LIN {X 0,Y 352.89,Z 1008.844,A -85,B 0,C 180,E1 14540.285,E2 14540.285} C_VEL
LIN {X 0,Y 348.435,Z 1029.036,A -85,B 0,C 180,E1 14538.872,E2 14538.872} C_VEL
LIN {X 0,Y 343.663,Z 1047.021,A -85,B 0,C 180,E1 14537.32,E2 14537.32} C_VEL
LIN {X 0,Y 338.159,Z 1064.954,A -85,B 0,C 180,E1 14535.444,E2 14535.444} C_VEL
LIN {X 0,Y 332.328,Z 1081.93,A -85,B 0,C 180,E1 14533.31,E2 14533.31} C_VEL
LIN {X 0,Y 326.202,Z 1097.954,A -85,B 0,C 180,E1 14530.873,E2 14530.873} C_VEL
LIN {X 0,Y 320.161,Z 1112.555,A -85,B 0,C 180,E1 14528.194,E2 14528.194} C_VEL
LIN {X 0,Y 314.194,Z 1126.284,A -85,B 0,C 180,E1 14525.168,E2 14525.168} C_VEL
LIN {X 0,Y 308.597,Z 1138.58,A -85,B 0,C 180,E1 14521.878,E2 14521.878} C_VEL
LIN {X 0,Y 303.562,Z 1149.432,A -85,B 0,C 180,E1 14518.313,E2 14518.313} C_VEL
LIN {X 0,Y 299.051,Z 1159.359,A -85,B 0,C 180,E1 14514.282,E2 14514.282} C_VEL
LIN {X 0,Y 295.723,Z 1167.059,A -85,B 0,C 180,E1 14510.38,E2 14510.38} C_VEL
LIN {X 0,Y 293.189,Z 1173.301,A -85,B 0,C 180,E1 14506.238,E2 14506.238} C_VEL
LIN {X 0,Y 291.464,Z 1178.188,A -85,B 0,C 180,E1 14501.878,E2 14501.878} C_VEL
LIN {X 0,Y 290.533,Z 1181.461,A -85,B 0,C 180,E1 14497.63,E2 14497.63} C_VEL
LIN {X 0,Y 290.087,Z 1183.156,A -85,B 0,C 180,E1 14493.557,E2 14493.557} C_VEL
LIN {X 0,Y 289.998,Z 1183.636,A -85,B 0,C 180,E1 14489.21,E2 14489.21} C_VEL
LIN {X 0,Y 290.174,Z 1182.841,A -85,B 0,C 180,E1 14485.257,E2 14485.257} C_VEL
LIN {X 0,Y 290.781,Z 1180.528,A -85,B 0,C 180,E1 14480.899,E2 14480.899} C_VEL
LIN {X 0,Y 291.906,Z 1176.965,A -85,B 0,C 180,E1 14476.733,E2 14476.733} C_VEL
LIN {X 0,Y 293.906,Z 1171.558,A -85,B 0,C 180,E1 14472.376,E2 14472.376} C_VEL
LIN {X 0,Y 296.703,Z 1164.7,A -85,B 0,C 180,E1 14468.243,E2 14468.243} C_VEL
LIN {X 0,Y 300.556,Z 1156.069,A -85,B 0,C 180,E1 14464.165,E2 14464.165} C_VEL
LIN {X 0,Y 305.239,Z 1146,A -85,B 0,C 180,E1 14460.356,E2 14460.356} C_VEL
LIN {X 0,Y 310.566,Z 1134.355,A -85,B 0,C 180,E1 14456.818,E2 14456.818} C_VEL
LIN {X 0,Y 316.433,Z 1121.267,A -85,B 0,C 180,E1 14453.557,E2 14453.557} C_VEL
LIN {X 0,Y 322.507,Z 1107.189,A -85,B 0,C 180,E1 14450.655,E2 14450.655} C_VEL
LIN {X 0,Y 328.545,Z 1092.152,A -85,B 0,C 180,E1 14448.089,E2 14448.089} C_VEL
LIN {X 0,Y 330.194,Z 1087.778,A -85,B 0,C 180,E1 14447.426,E2 14447.426} C_VEL
LIN {X 0,Y 331.529,Z 1082.425,A -85,B 0,C 180,E1 14446.505,E2 14446.505} C_VEL
LIN {X 0,Y 332.538,Z 1068.9,A -85,B 0,C 180,E1 14443.929,E2 14443.929} C_VEL
LIN {X 0,Y 333.902,Z 1062.973,A -85,B 0,C 180,E1 14443.095,E2 14443.095} C_VEL
LIN {X 0,Y 339.356,Z 1045.21,A -85,B 0,C 180,E1 14441.298,E2 14441.298} C_VEL
LIN {X 0,Y 344.539,Z 1025.743,A -85,B 0,C 180,E1 14439.676,E2 14439.676} C_VEL
LIN {X 0,Y 348.798,Z 1006.372,A -85,B 0,C 180,E1 14438.373,E2 14438.373} C_VEL
LIN {X 0,Y 352.358,Z 985.537,A -85,B 0,C 180,E1 14437.265,E2 14437.265} C_VEL
LIN {X 0,Y 355.126,Z 963.27,A -85,B 0,C 180,E1 14436.37,E2 14436.37} C_VEL
LIN {X 0,Y 356.788,Z 941.515,A -85,B 0,C 180,E1 14435.746,E2 14435.746} C_VEL
LIN {X 0,Y 365.568,Z 801.334,A -85,B 0,C 180,E1 14432.883,E2 14432.883} C_VEL
LIN {X 0,Y 356.931,Z 787.639,A -85,B 0,C 180,E1 14430.002,E2 14430.002} C_VEL
LIN {X 0,Y 349.574,Z 776.875,A -85,B 0,C 180,E1 14427.235,E2 14427.235} C_VEL
LIN {X 0,Y 343.426,Z 768.201,A -85,B 0,C 180,E1 14424.604,E2 14424.604} C_VEL
LIN {X 0,Y 339.11,Z 762.612,A -85,B 0,C 180,E1 14422.539,E2 14422.539} C_VEL
LIN {X 0,Y 335.486,Z 757.801,A -85,B 0,C 180,E1 14420.59,E2 14420.59} C_VEL
LIN {X 0,Y 331.948,Z 753.101,A -85,B 0,C 180,E1 14418.438,E2 14418.438} C_VEL
LIN {X 0,Y 328.093,Z 748.652,A -85,B 0,C 180,E1 14415.738,E2 14415.738} C_VEL
LIN {X 0,Y 327.083,Z 746.901,A -85,B 0,C 180,E1 14414.879,E2 14414.879} C_VEL
LIN {X 0,Y 323.777,Z 743.745,A -85,B 0,C 180,E1 14411.851,E2 14411.851} C_VEL
LIN {X 0,Y 322.352,Z 740.871,A -85,B 0,C 180,E1 14410.003,E2 14410.003} C_VEL
LIN {X 0,Y 318.916,Z 738.292,A -85,B 0,C 180,E1 14401.977,E2 14401.977} C_VEL
LIN {X 0,Y 319.479,Z 738.987,A -85,B 0,C 180,E1 14397.489,E2 14397.489} C_VEL
LIN {X 0,Y 322.551,Z 741.221,A -85,B 0,C 180,E1 14392.161,E2 14392.161} C_VEL
LIN {X 0,Y 324.789,Z 745.036,A -85,B 0,C 180,E1 14389.536,E2 14389.536} C_VEL
LIN {X 0,Y 325.775,Z 746.474,A -85,B 0,C 180,E1 14388.583,E2 14388.583} C_VEL
LIN {X 0,Y 329.072,Z 751.848,A -85,B 0,C 180,E1 14385.798,E2 14385.798} C_VEL
LIN {X 0,Y 332.186,Z 756.763,A -85,B 0,C 180,E1 14383.61,E2 14383.61} C_VEL
LIN {X 0,Y 337.821,Z 765.785,A -85,B 0,C 180,E1 14380.281,E2 14380.281} C_VEL
LIN {X 0,Y 345.029,Z 777.9,A -85,B 0,C 180,E1 14376.744,E2 14376.744} C_VEL
LIN {X 0,Y 351.975,Z 790.146,A -85,B 0,C 180,E1 14373.831,E2 14373.831} C_VEL
LIN {X 0,Y 359.361,Z 804.087,A -85,B 0,C 180,E1 14371.091,E2 14371.091} C_VEL
LIN {X 0,Y 365.817,Z 817.108,A -85,B 0,C 180,E1 14368.92,E2 14368.92} C_VEL
LIN {X 0,Y 356.497,Z 967.98,A -85,B 0,C 180,E1 14365.848,E2 14365.848} C_VEL
LIN {X 0,Y 352.635,Z 1028.021,A -85,B 0,C 180,E1 14364.593,E2 14364.593} C_VEL
LIN {X 0,Y 349.693,Z 1050.79,A -85,B 0,C 180,E1 14363.922,E2 14363.922} C_VEL
LIN {X 0,Y 345.509,Z 1072.869,A -85,B 0,C 180,E1 14363.073,E2 14363.073} C_VEL
LIN {X 0,Y 340.542,Z 1093.764,A -85,B 0,C 180,E1 14362.028,E2 14362.028} C_VEL
LIN {X 0,Y 334.973,Z 1113.773,A -85,B 0,C 180,E1 14360.721,E2 14360.721} C_VEL
LIN {X 0,Y 328.728,Z 1133.727,A -85,B 0,C 180,E1 14359.074,E2 14359.074} C_VEL
LIN {X 0,Y 322.404,Z 1152.314,A -85,B 0,C 180,E1 14357.187,E2 14357.187} C_VEL
LIN {X 0,Y 315.474,Z 1171.079,A -85,B 0,C 180,E1 14354.843,E2 14354.843} C_VEL
LIN {X 0,Y 308.833,Z 1188.354,A -85,B 0,C 180,E1 14352.204,E2 14352.204} C_VEL
LIN {X 0,Y 302.39,Z 1204.876,A -85,B 0,C 180,E1 14349.163,E2 14349.163} C_VEL
LIN {X 0,Y 296.695,Z 1219.605,A -85,B 0,C 180,E1 14345.899,E2 14345.899} C_VEL
LIN {X 0,Y 291.735,Z 1233.031,A -85,B 0,C 180,E1 14342.319,E2 14342.319} C_VEL
LIN {X 0,Y 287.46,Z 1245.829,A -85,B 0,C 180,E1 14338.231,E2 14338.231} C_VEL
LIN {X 0,Y 284.419,Z 1256.619,A -85,B 0,C 180,E1 14334.065,E2 14334.065} C_VEL
LIN {X 0,Y 282.517,Z 1265.437,A -85,B 0,C 180,E1 14329.861,E2 14329.861} C_VEL
LIN {X 0,Y 281.556,Z 1272.909,A -85,B 0,C 180,E1 14325.446,E2 14325.446} C_VEL
LIN {X 0,Y 281.384,Z 1278.064,A -85,B 0,C 180,E1 14321.477,E2 14321.477} C_VEL
LIN {X 0,Y 281.608,Z 1281.89,A -85,B 0,C 180,E1 14317.343,E2 14317.343} C_VEL
LIN {X 0,Y 281.909,Z 1283.834,A -85,B 0,C 180,E1 14313.864,E2 14313.864} C_VEL
LIN {X 0,Y 282.055,Z 1284.645,A -85,B 0,C 180,E1 14310.203,E2 14310.203} C_VEL
LIN {X 0,Y 281.933,Z 1283.994,A -85,B 0,C 180,E1 14306.544,E2 14306.544} C_VEL
LIN {X 0,Y 281.649,Z 1282.161,A -85,B 0,C 180,E1 14303.068,E2 14303.068} C_VEL
LIN {X 0,Y 281.387,Z 1278.535,A -85,B 0,C 180,E1 14298.938,E2 14298.938} C_VEL
LIN {X 0,Y 281.512,Z 1273.495,A -85,B 0,C 180,E1 14294.973,E2 14294.973} C_VEL
LIN {X 0,Y 282.383,Z 1266.228,A -85,B 0,C 180,E1 14290.56,E2 14290.56} C_VEL
LIN {X 0,Y 284.184,Z 1257.547,A -85,B 0,C 180,E1 14286.354,E2 14286.354} C_VEL
LIN {X 0,Y 287.105,Z 1246.946,A -85,B 0,C 180,E1 14282.183,E2 14282.183} C_VEL
LIN {X 0,Y 291.426,Z 1233.864,A -85,B 0,C 180,E1 14277.933,E2 14277.933} C_VEL
LIN {X 0,Y 296.389,Z 1220.386,A -85,B 0,C 180,E1 14274.296,E2 14274.296} C_VEL
LIN {X 0,Y 302.022,Z 1205.722,A -85,B 0,C 180,E1 14271.025,E2 14271.025} C_VEL
LIN {X 0,Y 308.619,Z 1188.814,A -85,B 0,C 180,E1 14267.885,E2 14267.885} C_VEL
LIN {X 0,Y 315.232,Z 1171.616,A -85,B 0,C 180,E1 14265.241,E2 14265.241} C_VEL
LIN {X 0,Y 321.854,Z 1153.662,A -85,B 0,C 180,E1 14262.982,E2 14262.982} C_VEL
LIN {X 0,Y 328.49,Z 1134.282,A -85,B 0,C 180,E1 14260.989,E2 14260.989} C_VEL
LIN {X 0,Y 334.765,Z 1114.287,A -85,B 0,C 180,E1 14259.327,E2 14259.327} C_VEL
LIN {X 0,Y 340.532,Z 1093.545,A -85,B 0,C 180,E1 14257.97,E2 14257.97} C_VEL
LIN {X 0,Y 345.5,Z 1072.584,A -85,B 0,C 180,E1 14256.924,E2 14256.924} C_VEL
LIN {X 0,Y 349.774,Z 1049.728,A -85,B 0,C 180,E1 14256.053,E2 14256.053} C_VEL
LIN {X 0,Y 352.628,Z 1027.173,A -85,B 0,C 180,E1 14255.396,E2 14255.396} C_VEL
LIN {X 0,Y 359.75,Z 913.323,A -85,B 0,C 180,E1 14253.052,E2 14253.052} C_VEL
LIN {X 0,Y 365.721,Z 817.058,A -85,B 0,C 180,E1 14251.089,E2 14251.089} C_VEL
LIN {X 0,Y 357.817,Z 801.163,A -85,B 0,C 180,E1 14248.407,E2 14248.407} C_VEL
LIN {X 0,Y 350.738,Z 788.072,A -85,B 0,C 180,E1 14245.736,E2 14245.736} C_VEL
LIN {X 0,Y 343.692,Z 775.733,A -85,B 0,C 180,E1 14242.717,E2 14242.717} C_VEL
LIN {X 0,Y 337.149,Z 764.789,A -85,B 0,C 180,E1 14239.444,E2 14239.444} C_VEL
LIN {X 0,Y 331.093,Z 755.02,A -85,B 0,C 180,E1 14235.77,E2 14235.77} C_VEL
LIN {X 0,Y 327.647,Z 749.717,A -85,B 0,C 180,E1 14233.23,E2 14233.23} C_VEL
LIN {X 0,Y 324.965,Z 745.249,A -85,B 0,C 180,E1 14230.817,E2 14230.817} C_VEL
LIN {X 0,Y 322.548,Z 741.379,A -85,B 0,C 180,E1 14228.108,E2 14228.108} C_VEL
LIN {X 0,Y 322.074,Z 740.745,A -85,B 0,C 180,E1 14227.492,E2 14227.492} C_VEL
LIN {X 0,Y 318.696,Z 738.017,A -85,B 0,C 180,E1 14219.64,E2 14219.64} C_VEL
LIN {X 0,Y 319.045,Z 738.532,A -85,B 0,C 180,E1 14215.686,E2 14215.686} C_VEL
LIN {X 0,Y 322.489,Z 741.155,A -85,B 0,C 180,E1 14209.459,E2 14209.459} C_VEL
LIN {X 0,Y 324.685,Z 744.973,A -85,B 0,C 180,E1 14206.918,E2 14206.918} C_VEL
LIN {X 0,Y 327.369,Z 747.393,A -85,B 0,C 180,E1 14204.635,E2 14204.635} C_VEL
LIN {X 0,Y 330.353,Z 751.615,A -85,B 0,C 180,E1 14202.382,E2 14202.382} C_VEL
LIN {X 0,Y 332.04,Z 753.353,A -85,B 0,C 180,E1 14201.294,E2 14201.294} C_VEL
LIN {X 0,Y 335.636,Z 757.967,A -85,B 0,C 180,E1 14199.146,E2 14199.146} C_VEL
LIN {X 0,Y 341,Z 765.139,A -85,B 0,C 180,E1 14196.361,E2 14196.361} C_VEL
LIN {X 0,Y 345.217,Z 770.847,A -85,B 0,C 180,E1 14194.434,E2 14194.434} C_VEL
LIN {X 0,Y 350.999,Z 778.969,A -85,B 0,C 180,E1 14192.057,E2 14192.057} C_VEL
LIN {X 0,Y 359.038,Z 790.932,A -85,B 0,C 180,E1 14189.129,E2 14189.129} C_VEL
LIN {X 0,Y 365.542,Z 801.506,A -85,B 0,C 180,E1 14186.993,E2 14186.993} C_VEL
LIN {X 0,Y 356.293,Z 947.507,A -85,B 0,C 180,E1 14184.004,E2 14184.004} C_VEL
LIN {X 0,Y 354.431,Z 969.192,A -85,B 0,C 180,E1 14183.324,E2 14183.324} C_VEL
LIN {X 0,Y 351.586,Z 990.18,A -85,B 0,C 180,E1 14182.413,E2 14182.413} C_VEL
LIN {X 0,Y 347.909,Z 1010.243,A -85,B 0,C 180,E1 14181.283,E2 14181.283} C_VEL
LIN {X 0,Y 343.562,Z 1029.462,A -85,B 0,C 180,E1 14179.941,E2 14179.941} C_VEL
LIN {X 0,Y 338.513,Z 1047.906,A -85,B 0,C 180,E1 14178.35,E2 14178.35} C_VEL
LIN {X 0,Y 332.67,Z 1066.352,A -85,B 0,C 180,E1 14176.412,E2 14176.412} C_VEL
LIN {X 0,Y 326.549,Z 1083.514,A -85,B 0,C 180,E1 14174.235,E2 14174.235} C_VEL
LIN {X 0,Y 320.261,Z 1099.348,A -85,B 0,C 180,E1 14171.801,E2 14171.801} C_VEL
LIN {X 0,Y 313.967,Z 1113.957,A -85,B 0,C 180,E1 14169.089,E2 14169.089} C_VEL
LIN {X 0,Y 307.655,Z 1127.852,A -85,B 0,C 180,E1 14165.978,E2 14165.978} C_VEL
LIN {X 0,Y 301.87,Z 1139.986,A -85,B 0,C 180,E1 14162.675,E2 14162.675} C_VEL
LIN {X 0,Y 296.579,Z 1150.838,A -85,B 0,C 180,E1 14159.042,E2 14159.042} C_VEL
LIN {X 0,Y 291.81,Z 1160.765,A -85,B 0,C 180,E1 14154.925,E2 14154.925} C_VEL
LIN {X 0,Y 288.272,Z 1168.465,A -85,B 0,C 180,E1 14150.931,E2 14150.931} C_VEL
LIN {X 0,Y 285.565,Z 1174.705,A -85,B 0,C 180,E1 14146.684,E2 14146.684} C_VEL
LIN {X 0,Y 283.709,Z 1179.588,A -85,B 0,C 180,E1 14142.207,E2 14142.207} C_VEL
LIN {X 0,Y 282.715,Z 1182.813,A -85,B 0,C 180,E1 14137.928,E2 14137.928} C_VEL
LIN {X 0,Y 282.217,Z 1184.547,A -85,B 0,C 180,E1 14133.656,E2 14133.656} C_VEL
LIN {X 0,Y 282.12,Z 1185.026,A -85,B 0,C 180,E1 14129.188,E2 14129.188} C_VEL
LIN {X 0,Y 282.313,Z 1184.233,A -85,B 0,C 180,E1 14125.124,E2 14125.124} C_VEL
LIN {X 0,Y 282.972,Z 1181.924,A -85,B 0,C 180,E1 14120.646,E2 14120.646} C_VEL
LIN {X 0,Y 284.187,Z 1178.365,A -85,B 0,C 180,E1 14116.366,E2 14116.366} C_VEL
LIN {X 0,Y 286.33,Z 1172.962,A -85,B 0,C 180,E1 14111.894,E2 14111.894} C_VEL
LIN {X 0,Y 289.32,Z 1166.104,A -85,B 0,C 180,E1 14107.658,E2 14107.658} C_VEL
LIN {X 0,Y 293.405,Z 1157.474,A -85,B 0,C 180,E1 14103.487,E2 14103.487} C_VEL
LIN {X 0,Y 298.34,Z 1147.404,A -85,B 0,C 180,E1 14099.599,E2 14099.599} C_VEL
LIN {X 0,Y 303.948,Z 1135.742,A -85,B 0,C 180,E1 14095.994,E2 14095.994} C_VEL
LIN {X 0,Y 310.08,Z 1122.666,A -85,B 0,C 180,E1 14092.686,E2 14092.686} C_VEL
LIN {X 0,Y 316.419,Z 1108.584,A -85,B 0,C 180,E1 14089.746,E2 14089.746} C_VEL
LIN {X 0,Y 322.699,Z 1093.545,A -85,B 0,C 180,E1 14087.15,E2 14087.15} C_VEL
LIN {X 0,Y 328.977,Z 1077.07,A -85,B 0,C 180,E1 14084.799,E2 14084.799} C_VEL
LIN {X 0,Y 333.902,Z 1062.973,A -85,B 0,C 180,E1 14083.095,E2 14083.095} C_VEL
LIN {X 0,Y 335.311,Z 1056.946,A -85,B 0,C 180,E1 14082.291,E2 14082.291} C_VEL
LIN {X 0,Y 336.215,Z 1041.964,A -85,B 0,C 180,E1 14080.007,E2 14080.007} C_VEL
LIN {X 0,Y 337.38,Z 1035.478,A -85,B 0,C 180,E1 14079.315,E2 14079.315} C_VEL
LIN {X 0,Y 342.109,Z 1016.487,A -85,B 0,C 180,E1 14077.9,E2 14077.9} C_VEL
LIN {X 0,Y 345.996,Z 997.035,A -85,B 0,C 180,E1 14076.741,E2 14076.741} C_VEL
LIN {X 0,Y 349.241,Z 975.642,A -85,B 0,C 180,E1 14075.743,E2 14075.743} C_VEL
LIN {X 0,Y 351.436,Z 954.76,A -85,B 0,C 180,E1 14075.015,E2 14075.015} C_VEL
LIN {X 0,Y 353.764,Z 917.385,A -85,B 0,C 180,E1 14074.155,E2 14074.155} C_VEL
LIN {X 0,Y 361.124,Z 805.509,A -85,B 0,C 180,E1 14071.88,E2 14071.88} C_VEL
LIN {X 0,Y 352.872,Z 792.375,A -85,B 0,C 180,E1 14068.982,E2 14068.982} C_VEL
LIN {X 0,Y 344.727,Z 780.224,A -85,B 0,C 180,E1 14065.698,E2 14065.698} C_VEL
LIN {X 0,Y 337.992,Z 770.862,A -85,B 0,C 180,E1 14062.526,E2 14062.526} C_VEL
LIN {X 0,Y 333.504,Z 765.063,A -85,B 0,C 180,E1 14060.077,E2 14060.077} C_VEL
LIN {X 0,Y 329.693,Z 760.015,A -85,B 0,C 180,E1 14057.654,E2 14057.654} C_VEL
LIN {X 0,Y 326.481,Z 756.026,A -85,B 0,C 180,E1 14055.271,E2 14055.271} C_VEL
LIN {X 0,Y 325.482,Z 754.519,A -85,B 0,C 180,E1 14054.408,E2 14054.408} C_VEL
LIN {X 0,Y 322.268,Z 751.064,A -85,B 0,C 180,E1 14051.272,E2 14051.272} C_VEL
LIN {X 0,Y 321.105,Z 748.705,A -85,B 0,C 180,E1 14049.68,E2 14049.68} C_VEL
LIN {X 0,Y 317.941,Z 746.234,A -85,B 0,C 180,E1 14041.983,E2 14041.983} C_VEL
LIN {X 0,Y 318.504,Z 746.942,A -85,B 0,C 180,E1 14037.481,E2 14037.481} C_VEL
LIN {X 0,Y 321.362,Z 749.076,A -85,B 0,C 180,E1 14032.402,E2 14032.402} C_VEL
LIN {X 0,Y 323.635,Z 752.927,A -85,B 0,C 180,E1 14029.678,E2 14029.678} C_VEL
LIN {X 0,Y 325.216,Z 755.754,A -85,B 0,C 180,E1 14028.113,E2 14028.113} C_VEL
LIN {X 0,Y 327.462,Z 759.302,A -85,B 0,C 180,E1 14026.222,E2 14026.222} C_VEL
LIN {X 0,Y 330.543,Z 764.349,A -85,B 0,C 180,E1 14023.977,E2 14023.977} C_VEL
LIN {X 0,Y 335.976,Z 773.309,A -85,B 0,C 180,E1 14020.666,E2 14020.666} C_VEL
LIN {X 0,Y 342.612,Z 784.779,A -85,B 0,C 180,E1 14017.298,E2 14017.298} C_VEL
LIN {X 0,Y 349.295,Z 796.876,A -85,B 0,C 180,E1 14014.391,E2 14014.391} C_VEL
LIN {X 0,Y 356.412,Z 810.672,A -85,B 0,C 180,E1 14011.654,E2 14011.654} C_VEL
LIN {X 0,Y 361.421,Z 821.196,A -85,B 0,C 180,E1 14009.887,E2 14009.887} C_VEL
LIN {X 0,Y 348.204,Z 1024.194,A -85,B 0,C 180,E1 14005.738,E2 14005.738} C_VEL
LIN {X 0,Y 345.397,Z 1046.631,A -85,B 0,C 180,E1 14005.1,E2 14005.1} C_VEL
LIN {X 0,Y 341.208,Z 1069.196,A -85,B 0,C 180,E1 14004.26,E2 14004.26} C_VEL
LIN {X 0,Y 336.237,Z 1089.948,A -85,B 0,C 180,E1 14003.262,E2 14003.262} C_VEL
LIN {X 0,Y 330.546,Z 1109.941,A -85,B 0,C 180,E1 14001.995,E2 14001.995} C_VEL
LIN {X 0,Y 323.709,Z 1131.293,A -85,B 0,C 180,E1 14000.271,E2 14000.271} C_VEL
LIN {X 0,Y 317.051,Z 1150.222,A -85,B 0,C 180,E1 13998.364,E2 13998.364} C_VEL
LIN {X 0,Y 309.857,Z 1168.972,A -85,B 0,C 180,E1 13996.018,E2 13996.018} C_VEL
LIN {X 0,Y 302.883,Z 1186.338,A -85,B 0,C 180,E1 13993.363,E2 13993.363} C_VEL
LIN {X 0,Y 296.281,Z 1202.484,A -85,B 0,C 180,E1 13990.385,E2 13990.385} C_VEL
LIN {X 0,Y 290.223,Z 1217.286,A -85,B 0,C 180,E1 13987.076,E2 13987.076} C_VEL
LIN {X 0,Y 284.73,Z 1231.282,A -85,B 0,C 180,E1 13983.306,E2 13983.306} C_VEL
LIN {X 0,Y 280.255,Z 1243.769,A -85,B 0,C 180,E1 13979.259,E2 13979.259} C_VEL
LIN {X 0,Y 276.924,Z 1254.627,A -85,B 0,C 180,E1 13974.988,E2 13974.988} C_VEL
LIN {X 0,Y 274.799,Z 1263.568,A -85,B 0,C 180,E1 13970.666,E2 13970.666} C_VEL
LIN {X 0,Y 273.67,Z 1271.159,A -85,B 0,C 180,E1 13966.12,E2 13966.12} C_VEL
LIN {X 0,Y 273.441,Z 1276.389,A -85,B 0,C 180,E1 13962.03,E2 13962.03} C_VEL
LIN {X 0,Y 273.659,Z 1280.338,A -85,B 0,C 180,E1 13957.769,E2 13957.769} C_VEL
LIN {X 0,Y 273.999,Z 1282.355,A -85,B 0,C 180,E1 13954.185,E2 13954.185} C_VEL
LIN {X 0,Y 274.169,Z 1283.18,A -85,B 0,C 180,E1 13950.836,E2 13950.836} C_VEL
LIN {X 0,Y 274.077,Z 1282.839,A -85,B 0,C 180,E1 13947.073,E2 13947.073} C_VEL
LIN {X 0,Y 273.767,Z 1281.029,A -85,B 0,C 180,E1 13943.289,E2 13943.289} C_VEL
LIN {X 0,Y 273.465,Z 1277.766,A -85,B 0,C 180,E1 13939.254,E2 13939.254} C_VEL
LIN {X 0,Y 273.557,Z 1272.643,A -85,B 0,C 180,E1 13934.96,E2 13934.96} C_VEL
LIN {X 0,Y 274.364,Z 1265.972,A -85,B 0,C 180,E1 13930.633,E2 13930.633} C_VEL
LIN {X 0,Y 276.17,Z 1257.449,A -85,B 0,C 180,E1 13926.306,E2 13926.306} C_VEL
LIN {X 0,Y 279.311,Z 1246.603,A -85,B 0,C 180,E1 13921.803,E2 13921.803} C_VEL
LIN {X 0,Y 283.361,Z 1234.976,A -85,B 0,C 180,E1 13917.805,E2 13917.805} C_VEL
LIN {X 0,Y 288.625,Z 1221.215,A -85,B 0,C 180,E1 13913.921,E2 13913.921} C_VEL
LIN {X 0,Y 294.763,Z 1206.044,A -85,B 0,C 180,E1 13910.38,E2 13910.38} C_VEL
LIN {X 0,Y 301.363,Z 1190.014,A -85,B 0,C 180,E1 13907.276,E2 13907.276} C_VEL
LIN {X 0,Y 308.16,Z 1173.152,A -85,B 0,C 180,E1 13904.58,E2 13904.58} C_VEL
LIN {X 0,Y 315.186,Z 1154.974,A -85,B 0,C 180,E1 13902.209,E2 13902.209} C_VEL
LIN {X 0,Y 322.281,Z 1135.335,A -85,B 0,C 180,E1 13900.117,E2 13900.117} C_VEL
LIN {X 0,Y 328.766,Z 1115.703,A -85,B 0,C 180,E1 13898.434,E2 13898.434} C_VEL
LIN {X 0,Y 334.613,Z 1095.56,A -85,B 0,C 180,E1 13897.08,E2 13897.08} C_VEL
LIN {X 0,Y 340.185,Z 1073.394,A -85,B 0,C 180,E1 13895.932,E2 13895.932} C_VEL
LIN {X 0,Y 344.585,Z 1051.413,A -85,B 0,C 180,E1 13895.066,E2 13895.066} C_VEL
LIN {X 0,Y 347.631,Z 1028.996,A -85,B 0,C 180,E1 13894.394,E2 13894.394} C_VEL
LIN {X 0,Y 350.084,Z 995.699,A -85,B 0,C 180,E1 13893.665,E2 13893.665} C_VEL
LIN {X 0,Y 361.293,Z 820.87,A -85,B 0,C 180,E1 13890.106,E2 13890.106} C_VEL
LIN {X 0,Y 353.804,Z 805.57,A -85,B 0,C 180,E1 13887.428,E2 13887.428} C_VEL
LIN {X 0,Y 346.866,Z 792.534,A -85,B 0,C 180,E1 13884.661,E2 13884.661} C_VEL
LIN {X 0,Y 340.077,Z 780.45,A -85,B 0,C 180,E1 13881.562,E2 13881.562} C_VEL
LIN {X 0,Y 334.728,Z 771.416,A -85,B 0,C 180,E1 13878.73,E2 13878.73} C_VEL
LIN {X 0,Y 329.477,Z 762.556,A -85,B 0,C 180,E1 13875.398,E2 13875.398} C_VEL
LIN {X 0,Y 326.023,Z 757.116,A -85,B 0,C 180,E1 13872.756,E2 13872.756} C_VEL
LIN {X 0,Y 323.623,Z 752.949,A -85,B 0,C 180,E1 13870.503,E2 13870.503} C_VEL
LIN {X 0,Y 321.233,Z 748.915,A -85,B 0,C 180,E1 13867.691,E2 13867.691} C_VEL
LIN {X 0,Y 317.751,Z 746.016,A -85,B 0,C 180,E1 13860,E2 13860} C_VEL
LIN {X 0,Y 317.91,Z 746.263,A -85,B 0,C 180,E1 13856.393,E2 13856.393} C_VEL
LIN {X 0,Y 321.298,Z 749.039,A -85,B 0,C 180,E1 13849.692,E2 13849.692} C_VEL
LIN {X 0,Y 323.447,Z 752.777,A -85,B 0,C 180,E1 13847.14,E2 13847.14} C_VEL
LIN {X 0,Y 325.919,Z 755.057,A -85,B 0,C 180,E1 13844.975,E2 13844.975} C_VEL
LIN {X 0,Y 328.951,Z 759.365,A -85,B 0,C 180,E1 13842.628,E2 13842.628} C_VEL
LIN {X 0,Y 330.476,Z 761.049,A -85,B 0,C 180,E1 13841.614,E2 13841.614} C_VEL
LIN {X 0,Y 334.864,Z 766.905,A -85,B 0,C 180,E1 13838.958,E2 13838.958} C_VEL
LIN {X 0,Y 339.197,Z 772.762,A -85,B 0,C 180,E1 13836.688,E2 13836.688} C_VEL
LIN {X 0,Y 344.785,Z 780.37,A -85,B 0,C 180,E1 13834.123,E2 13834.123} C_VEL
LIN {X 0,Y 353.678,Z 793.642,A -85,B 0,C 180,E1 13830.58,E2 13830.58} C_VEL
LIN {X 0,Y 361.1,Z 805.724,A -85,B 0,C 180,E1 13827.99,E2 13827.99} C_VEL
LIN {X 0,Y 351.736,Z 948.502,A -85,B 0,C 180,E1 13825.057,E2 13825.057} C_VEL
LIN {X 0,Y 349.827,Z 970.215,A -85,B 0,C 180,E1 13824.375,E2 13824.375} C_VEL
LIN {X 0,Y 346.884,Z 991.265,A -85,B 0,C 180,E1 13823.46,E2 13823.46} C_VEL
LIN {X 0,Y 343.038,Z 1011.641,A -85,B 0,C 180,E1 13822.309,E2 13822.309} C_VEL
LIN {X 0,Y 338.545,Z 1030.859,A -85,B 0,C 180,E1 13820.961,E2 13820.961} C_VEL
LIN {X 0,Y 333.333,Z 1049.278,A -85,B 0,C 180,E1 13819.365,E2 13819.365} C_VEL
LIN {X 0,Y 327.279,Z 1067.749,A -85,B 0,C 180,E1 13817.413,E2 13817.413} C_VEL
LIN {X 0,Y 321.012,Z 1084.726,A -85,B 0,C 180,E1 13815.246,E2 13815.246} C_VEL
LIN {X 0,Y 314.622,Z 1100.229,A -85,B 0,C 180,E1 13812.849,E2 13812.849} C_VEL
LIN {X 0,Y 307.854,Z 1115.359,A -85,B 0,C 180,E1 13810.02,E2 13810.02} C_VEL
LIN {X 0,Y 301.332,Z 1129.121,A -85,B 0,C 180,E1 13806.901,E2 13806.901} C_VEL
LIN {X 0,Y 295.206,Z 1141.392,A -85,B 0,C 180,E1 13803.509,E2 13803.509} C_VEL
LIN {X 0,Y 289.644,Z 1152.245,A -85,B 0,C 180,E1 13799.807,E2 13799.807} C_VEL
LIN {X 0,Y 284.605,Z 1162.173,A -85,B 0,C 180,E1 13795.601,E2 13795.601} C_VEL
LIN {X 0,Y 280.852,Z 1169.871,A -85,B 0,C 180,E1 13791.511,E2 13791.511} C_VEL
LIN {X 0,Y 277.957,Z 1176.109,A -85,B 0,C 180,E1 13787.155,E2 13787.155} C_VEL
LIN {X 0,Y 275.964,Z 1180.988,A -85,B 0,C 180,E1 13782.555,E2 13782.555} C_VEL
LIN {X 0,Y 274.887,Z 1184.209,A -85,B 0,C 180,E1 13778.155,E2 13778.155} C_VEL
LIN {X 0,Y 274.348,Z 1185.939,A -85,B 0,C 180,E1 13773.761,E2 13773.761} C_VEL
LIN {X 0,Y 274.242,Z 1186.417,A -85,B 0,C 180,E1 13769.164,E2 13769.164} C_VEL
LIN {X 0,Y 274.452,Z 1185.625,A -85,B 0,C 180,E1 13764.984,E2 13764.984} C_VEL
LIN {X 0,Y 275.167,Z 1183.32,A -85,B 0,C 180,E1 13760.378,E2 13760.378} C_VEL
LIN {X 0,Y 276.476,Z 1179.766,A -85,B 0,C 180,E1 13755.978,E2 13755.978} C_VEL
LIN {X 0,Y 278.647,Z 1174.633,A -85,B 0,C 180,E1 13751.593,E2 13751.593} C_VEL
LIN {X 0,Y 281.79,Z 1167.874,A -85,B 0,C 180,E1 13747.248,E2 13747.248} C_VEL
LIN {X 0,Y 285.952,Z 1159.588,A -85,B 0,C 180,E1 13743.08,E2 13743.08} C_VEL
LIN {X 0,Y 290.93,Z 1149.874,A -85,B 0,C 180,E1 13739.199,E2 13739.199} C_VEL
LIN {X 0,Y 296.711,Z 1138.458,A -85,B 0,C 180,E1 13735.521,E2 13735.521} C_VEL
LIN {X 0,Y 303.053,Z 1125.647,A -85,B 0,C 180,E1 13732.146,E2 13732.146} C_VEL
LIN {X 0,Y 309.793,Z 1111.407,A -85,B 0,C 180,E1 13729.068,E2 13729.068} C_VEL
LIN {X 0,Y 316.525,Z 1095.904,A -85,B 0,C 180,E1 13726.335,E2 13726.335} C_VEL
LIN {X 0,Y 323.231,Z 1079.068,A -85,B 0,C 180,E1 13723.886,E2 13723.886} C_VEL
LIN {X 0,Y 329.376,Z 1061.96,A -85,B 0,C 180,E1 13721.822,E2 13721.822} C_VEL
LIN {X 0,Y 334.988,Z 1043.996,A -85,B 0,C 180,E1 13720.043,E2 13720.043} C_VEL
LIN {X 0,Y 337.38,Z 1035.478,A -85,B 0,C 180,E1 13719.315,E2 13719.315} C_VEL
LIN {X 0,Y 338.592,Z 1028.887,A -85,B 0,C 180,E1 13718.645,E2 13718.645} C_VEL
LIN {X 0,Y 339.096,Z 1012.653,A -85,B 0,C 180,E1 13716.637,E2 13716.637} C_VEL
LIN {X 0,Y 339.952,Z 1005.7,A -85,B 0,C 180,E1 13716.083,E2 13716.083} C_VEL
LIN {X 0,Y 343.561,Z 985.118,A -85,B 0,C 180,E1 13715.02,E2 13715.02} C_VEL
LIN {X 0,Y 346.205,Z 963.954,A -85,B 0,C 180,E1 13714.195,E2 13714.195} C_VEL
LIN {X 0,Y 347.99,Z 940.649,A -85,B 0,C 180,E1 13713.548,E2 13713.548} C_VEL
LIN {X 0,Y 356.777,Z 809.833,A -85,B 0,C 180,E1 13710.854,E2 13710.854} C_VEL
LIN {X 0,Y 349.5,Z 798.065,A -85,B 0,C 180,E1 13708.167,E2 13708.167} C_VEL
LIN {X 0,Y 342.23,Z 787.038,A -85,B 0,C 180,E1 13705.111,E2 13705.111} C_VEL
LIN {X 0,Y 335.916,Z 778.069,A -85,B 0,C 180,E1 13702.027,E2 13702.027} C_VEL
LIN {X 0,Y 331.69,Z 772.464,A -85,B 0,C 180,E1 13699.64,E2 13699.64} C_VEL
LIN {X 0,Y 328.105,Z 767.601,A -85,B 0,C 180,E1 13697.285,E2 13697.285} C_VEL
LIN {X 0,Y 324.89,Z 763.4,A -85,B 0,C 180,E1 13694.8,E2 13694.8} C_VEL
LIN {X 0,Y 324.109,Z 762.262,A -85,B 0,C 180,E1 13694.106,E2 13694.106} C_VEL
LIN {X 0,Y 320.997,Z 758.758,A -85,B 0,C 180,E1 13690.953,E2 13690.953} C_VEL
LIN {X 0,Y 320.003,Z 756.6,A -85,B 0,C 180,E1 13689.532,E2 13689.532} C_VEL
LIN {X 0,Y 316.967,Z 754.176,A -85,B 0,C 180,E1 13681.989,E2 13681.989} C_VEL
LIN {X 0,Y 317.472,Z 754.834,A -85,B 0,C 180,E1 13677.654,E2 13677.654} C_VEL
LIN {X 0,Y 320.18,Z 756.923,A -85,B 0,C 180,E1 13672.644,E2 13672.644} C_VEL
LIN {X 0,Y 322.483,Z 760.818,A -85,B 0,C 180,E1 13669.821,E2 13669.821} C_VEL
LIN {X 0,Y 326.025,Z 767.05,A -85,B 0,C 180,E1 13666.522,E2 13666.522} C_VEL
LIN {X 0,Y 328.855,Z 771.819,A -85,B 0,C 180,E1 13664.391,E2 13664.391} C_VEL
LIN {X 0,Y 334.146,Z 780.832,A -85,B 0,C 180,E1 13661.055,E2 13661.055} C_VEL
LIN {X 0,Y 340.389,Z 791.976,A -85,B 0,C 180,E1 13657.779,E2 13657.779} C_VEL
LIN {X 0,Y 346.649,Z 803.604,A -85,B 0,C 180,E1 13654.959,E2 13654.959} C_VEL
LIN {X 0,Y 353.597,Z 817.449,A -85,B 0,C 180,E1 13652.189,E2 13652.189} C_VEL
LIN {X 0,Y 357.053,Z 825.011,A -85,B 0,C 180,E1 13650.908,E2 13650.908} C_VEL
LIN {X 0,Y 343.648,Z 1023.437,A -85,B 0,C 180,E1 13646.841,E2 13646.841} C_VEL
LIN {X 0,Y 340.733,Z 1045.78,A -85,B 0,C 180,E1 13646.2,E2 13646.2} C_VEL
LIN {X 0,Y 336.33,Z 1068.676,A -85,B 0,C 180,E1 13645.342,E2 13645.342} C_VEL
LIN {X 0,Y 331.099,Z 1089.75,A -85,B 0,C 180,E1 13644.322,E2 13644.322} C_VEL
LIN {X 0,Y 324.935,Z 1110.558,A -85,B 0,C 180,E1 13642.985,E2 13642.985} C_VEL
LIN {X 0,Y 318.201,Z 1130.679,A -85,B 0,C 180,E1 13641.336,E2 13641.336} C_VEL
LIN {X 0,Y 311.038,Z 1150.152,A -85,B 0,C 180,E1 13639.342,E2 13639.342} C_VEL
LIN {X 0,Y 303.912,Z 1168.033,A -85,B 0,C 180,E1 13637.077,E2 13637.077} C_VEL
LIN {X 0,Y 296.619,Z 1185.367,A -85,B 0,C 180,E1 13634.389,E2 13634.389} C_VEL
LIN {X 0,Y 289.506,Z 1201.904,A -85,B 0,C 180,E1 13631.272,E2 13631.272} C_VEL
LIN {X 0,Y 283.192,Z 1216.63,A -85,B 0,C 180,E1 13627.902,E2 13627.902} C_VEL
LIN {X 0,Y 277.596,Z 1230.051,A -85,B 0,C 180,E1 13624.185,E2 13624.185} C_VEL
LIN {X 0,Y 272.716,Z 1242.855,A -85,B 0,C 180,E1 13619.908,E2 13619.908} C_VEL
LIN {X 0,Y 269.182,Z 1253.714,A -85,B 0,C 180,E1 13615.498,E2 13615.498} C_VEL
LIN {X 0,Y 266.945,Z 1262.506,A -85,B 0,C 180,E1 13611.073,E2 13611.073} C_VEL
LIN {X 0,Y 265.715,Z 1270.309,A -85,B 0,C 180,E1 13606.167,E2 13606.167} C_VEL
LIN {X 0,Y 265.508,Z 1275.691,A -85,B 0,C 180,E1 13601.733,E2 13601.733} C_VEL
LIN {X 0,Y 265.794,Z 1279.35,A -85,B 0,C 180,E1 13597.348,E2 13597.348} C_VEL
LIN {X 0,Y 266.146,Z 1281.206,A -85,B 0,C 180,E1 13593.662,E2 13593.662} C_VEL
LIN {X 0,Y 266.298,Z 1281.863,A -85,B 0,C 180,E1 13589.785,E2 13589.785} C_VEL
LIN {X 0,Y 266.131,Z 1281.119,A -85,B 0,C 180,E1 13586.122,E2 13586.122} C_VEL
LIN {X 0,Y 265.773,Z 1279.2,A -85,B 0,C 180,E1 13582.434,E2 13582.434} C_VEL
LIN {X 0,Y 265.505,Z 1275.432,A -85,B 0,C 180,E1 13578.047,E2 13578.047} C_VEL
LIN {X 0,Y 265.716,Z 1270.296,A -85,B 0,C 180,E1 13573.833,E2 13573.833} C_VEL
LIN {X 0,Y 266.862,Z 1262.891,A -85,B 0,C 180,E1 13569.15,E2 13569.15} C_VEL
LIN {X 0,Y 269.055,Z 1254.126,A -85,B 0,C 180,E1 13564.701,E2 13564.701} C_VEL
LIN {X 0,Y 272.508,Z 1243.394,A -85,B 0,C 180,E1 13560.31,E2 13560.31} C_VEL
LIN {X 0,Y 277.33,Z 1230.677,A -85,B 0,C 180,E1 13556.018,E2 13556.018} C_VEL
LIN {X 0,Y 282.845,Z 1217.401,A -85,B 0,C 180,E1 13552.299,E2 13552.299} C_VEL
LIN {X 0,Y 289.104,Z 1202.741,A -85,B 0,C 180,E1 13548.922,E2 13548.922} C_VEL
LIN {X 0,Y 296.372,Z 1185.844,A -85,B 0,C 180,E1 13545.707,E2 13545.707} C_VEL
LIN {X 0,Y 303.607,Z 1168.663,A -85,B 0,C 180,E1 13543.023,E2 13543.023} C_VEL
LIN {X 0,Y 310.756,Z 1150.72,A -85,B 0,C 180,E1 13540.738,E2 13540.738} C_VEL
LIN {X 0,Y 317.895,Z 1131.356,A -85,B 0,C 180,E1 13538.74,E2 13538.74} C_VEL
LIN {X 0,Y 324.611,Z 1111.379,A -85,B 0,C 180,E1 13537.085,E2 13537.085} C_VEL
LIN {X 0,Y 330.753,Z 1090.655,A -85,B 0,C 180,E1 13535.743,E2 13535.743} C_VEL
LIN {X 0,Y 336.057,Z 1069.496,A -85,B 0,C 180,E1 13534.705,E2 13534.705} C_VEL
LIN {X 0,Y 340.549,Z 1046.388,A -85,B 0,C 180,E1 13533.831,E2 13533.831} C_VEL
LIN {X 0,Y 343.499,Z 1024.073,A -85,B 0,C 180,E1 13533.185,E2 13533.185} C_VEL
LIN {X 0,Y 352.35,Z 892.553,A -85,B 0,C 180,E1 13530.467,E2 13530.467} C_VEL
LIN {X 0,Y 356.921,Z 824.582,A -85,B 0,C 180,E1 13529.08,E2 13529.08} C_VEL
LIN {X 0,Y 349.787,Z 809.91,A -85,B 0,C 180,E1 13526.391,E2 13526.391} C_VEL
LIN {X 0,Y 343.312,Z 797.437,A -85,B 0,C 180,E1 13523.652,E2 13523.652} C_VEL
LIN {X 0,Y 337.517,Z 786.953,A -85,B 0,C 180,E1 13520.868,E2 13520.868} C_VEL
LIN {X 0,Y 332.715,Z 778.558,A -85,B 0,C 180,E1 13518.212,E2 13518.212} C_VEL
LIN {X 0,Y 327.754,Z 769.932,A -85,B 0,C 180,E1 13514.938,E2 13514.938} C_VEL
LIN {X 0,Y 324.522,Z 764.657,A -85,B 0,C 180,E1 13512.364,E2 13512.364} C_VEL
LIN {X 0,Y 322.29,Z 760.647,A -85,B 0,C 180,E1 13510.185,E2 13510.185} C_VEL
LIN {X 0,Y 319.853,Z 756.524,A -85,B 0,C 180,E1 13507.183,E2 13507.183} C_VEL
LIN {X 0,Y 316.745,Z 753.903,A -85,B 0,C 180,E1 13499.638,E2 13499.638} C_VEL
LIN {X 0,Y 317.052,Z 754.385,A -85,B 0,C 180,E1 13495.84,E2 13495.84} C_VEL
LIN {X 0,Y 320.114,Z 756.908,A -85,B 0,C 180,E1 13489.926,E2 13489.926} C_VEL
LIN {X 0,Y 322.478,Z 760.875,A -85,B 0,C 180,E1 13487.1,E2 13487.1} C_VEL
LIN {X 0,Y 324.529,Z 762.81,A -85,B 0,C 180,E1 13485.275,E2 13485.275} C_VEL
LIN {X 0,Y 327.688,Z 767.243,A -85,B 0,C 180,E1 13482.784,E2 13482.784} C_VEL
LIN {X 0,Y 329.043,Z 768.942,A -85,B 0,C 180,E1 13481.852,E2 13481.852} C_VEL
LIN {X 0,Y 333.153,Z 774.506,A -85,B 0,C 180,E1 13479.305,E2 13479.305} C_VEL
LIN {X 0,Y 337.326,Z 780.261,A -85,B 0,C 180,E1 13477.059,E2 13477.059} C_VEL
LIN {X 0,Y 342.545,Z 787.55,A -85,B 0,C 180,E1 13474.591,E2 13474.591} C_VEL
LIN {X 0,Y 351.065,Z 800.555,A -85,B 0,C 180,E1 13471.088,E2 13471.088} C_VEL
LIN {X 0,Y 356.758,Z 810.124,A -85,B 0,C 180,E1 13469.008,E2 13469.008} C_VEL
LIN {X 0,Y 347.316,Z 949.287,A -85,B 0,C 180,E1 13466.142,E2 13466.142} C_VEL
LIN {X 0,Y 345.376,Z 970.984,A -85,B 0,C 180,E1 13465.465,E2 13465.465} C_VEL
LIN {X 0,Y 342.316,Z 992.245,A -85,B 0,C 180,E1 13464.541,E2 13464.541} C_VEL
LIN {X 0,Y 338.279,Z 1013.041,A -85,B 0,C 180,E1 13463.365,E2 13463.365} C_VEL
LIN {X 0,Y 333.639,Z 1032.255,A -85,B 0,C 180,E1 13462.012,E2 13462.012} C_VEL
LIN {X 0,Y 328.253,Z 1050.675,A -85,B 0,C 180,E1 13460.409,E2 13460.409} C_VEL
LIN {X 0,Y 321.991,Z 1069.146,A -85,B 0,C 180,E1 13458.447,E2 13458.447} C_VEL
LIN {X 0,Y 315.5,Z 1086.125,A -85,B 0,C 180,E1 13456.264,E2 13456.264} C_VEL
LIN {X 0,Y 308.867,Z 1101.629,A -85,B 0,C 180,E1 13453.847,E2 13453.847} C_VEL
LIN {X 0,Y 301.825,Z 1116.761,A -85,B 0,C 180,E1 13450.988,E2 13450.988} C_VEL
LIN {X 0,Y 295.032,Z 1130.497,A -85,B 0,C 180,E1 13447.835,E2 13447.835} C_VEL
LIN {X 0,Y 288.607,Z 1142.798,A -85,B 0,C 180,E1 13444.38,E2 13444.38} C_VEL
LIN {X 0,Y 282.765,Z 1153.652,A -85,B 0,C 180,E1 13440.609,E2 13440.609} C_VEL
LIN {X 0,Y 277.44,Z 1163.58,A -85,B 0,C 180,E1 13436.312,E2 13436.312} C_VEL
LIN {X 0,Y 273.457,Z 1171.278,A -85,B 0,C 180,E1 13432.123,E2 13432.123} C_VEL
LIN {X 0,Y 270.376,Z 1177.513,A -85,B 0,C 180,E1 13427.652,E2 13427.652} C_VEL
LIN {X 0,Y 268.229,Z 1182.388,A -85,B 0,C 180,E1 13422.924,E2 13422.924} C_VEL
LIN {X 0,Y 267.062,Z 1185.604,A -85,B 0,C 180,E1 13418.396,E2 13418.396} C_VEL
LIN {X 0,Y 266.48,Z 1187.331,A -85,B 0,C 180,E1 13413.872,E2 13413.872} C_VEL
LIN {X 0,Y 266.364,Z 1187.807,A -85,B 0,C 180,E1 13409.14,E2 13409.14} C_VEL
LIN {X 0,Y 266.592,Z 1187.017,A -85,B 0,C 180,E1 13404.836,E2 13404.836} C_VEL
LIN {X 0,Y 267.366,Z 1184.716,A -85,B 0,C 180,E1 13400.095,E2 13400.095} C_VEL
LIN {X 0,Y 268.776,Z 1181.167,A -85,B 0,C 180,E1 13395.568,E2 13395.568} C_VEL
LIN {X 0,Y 271.107,Z 1176.037,A -85,B 0,C 180,E1 13391.062,E2 13391.062} C_VEL
LIN {X 0,Y 274.465,Z 1169.278,A -85,B 0,C 180,E1 13386.605,E2 13386.605} C_VEL
LIN {X 0,Y 278.901,Z 1160.934,A -85,B 0,C 180,E1 13382.313,E2 13382.313} C_VEL
LIN {X 0,Y 284.414,Z 1150.752,A -85,B 0,C 180,E1 13378.176,E2 13378.176} C_VEL
LIN {X 0,Y 290.19,Z 1139.86,A -85,B 0,C 180,E1 13374.632,E2 13374.632} C_VEL
LIN {X 0,Y 296.823,Z 1127.046,A -85,B 0,C 180,E1 13371.206,E2 13371.206} C_VEL
LIN {X 0,Y 303.85,Z 1112.803,A -85,B 0,C 180,E1 13368.089,E2 13368.089} C_VEL
LIN {X 0,Y 310.575,Z 1097.91,A -85,B 0,C 180,E1 13365.428,E2 13365.428} C_VEL
LIN {X 0,Y 317.558,Z 1081.095,A -85,B 0,C 180,E1 13362.944,E2 13362.944} C_VEL
LIN {X 0,Y 323.913,Z 1064.124,A -85,B 0,C 180,E1 13360.866,E2 13360.866} C_VEL
LIN {X 0,Y 329.972,Z 1045.381,A -85,B 0,C 180,E1 13358.995,E2 13358.995} C_VEL
LIN {X 0,Y 335.389,Z 1025.719,A -85,B 0,C 180,E1 13357.396,E2 13357.396} C_VEL
LIN {X 0,Y 339.952,Z 1005.7,A -85,B 0,C 180,E1 13356.083,E2 13356.083} C_VEL
LIN {X 0,Y 340.82,Z 998.628,A -85,B 0,C 180,E1 13355.561,E2 13355.561} C_VEL
LIN {X 0,Y 340.479,Z 981.246,A -85,B 0,C 180,E1 13353.862,E2 13353.862} C_VEL
LIN {X 0,Y 340.854,Z 974.003,A -85,B 0,C 180,E1 13353.407,E2 13353.407} C_VEL
LIN {X 0,Y 342.981,Z 952.155,A -85,B 0,C 180,E1 13352.7,E2 13352.7} C_VEL
LIN {X 0,Y 347.216,Z 890.32,A -85,B 0,C 180,E1 13351.374,E2 13351.374} C_VEL
LIN {X 0,Y 352.634,Z 814.248,A -85,B 0,C 180,E1 13349.833,E2 13349.833} C_VEL
LIN {X 0,Y 345.362,Z 802.431,A -85,B 0,C 180,E1 13346.989,E2 13346.989} C_VEL
LIN {X 0,Y 338.672,Z 792.285,A -85,B 0,C 180,E1 13343.997,E2 13343.997} C_VEL
LIN {X 0,Y 333.41,Z 784.728,A -85,B 0,C 180,E1 13341.277,E2 13341.277} C_VEL
LIN {X 0,Y 329.896,Z 779.861,A -85,B 0,C 180,E1 13339.199,E2 13339.199} C_VEL
LIN {X 0,Y 326.531,Z 775.184,A -85,B 0,C 180,E1 13336.912,E2 13336.912} C_VEL
LIN {X 0,Y 323.321,Z 770.772,A -85,B 0,C 180,E1 13334.324,E2 13334.324} C_VEL
LIN {X 0,Y 322.161,Z 769.536,A -85,B 0,C 180,E1 13333.278,E2 13333.278} C_VEL
LIN {X 0,Y 319.418,Z 765.785,A -85,B 0,C 180,E1 13330.187,E2 13330.187} C_VEL
LIN {X 0,Y 318.77,Z 764.434,A -85,B 0,C 180,E1 13329.205,E2 13329.205} C_VEL
LIN {X 0,Y 315.982,Z 762.1,A -85,B 0,C 180,E1 13321.814,E2 13321.814} C_VEL
LIN {X 0,Y 316.552,Z 762.853,A -85,B 0,C 180,E1 13317.466,E2 13317.466} C_VEL
LIN {X 0,Y 319.004,Z 764.764,A -85,B 0,C 180,E1 13312.889,E2 13312.889} C_VEL
LIN {X 0,Y 321.639,Z 769.455,A -85,B 0,C 180,E1 13309.613,E2 13309.613} C_VEL
LIN {X 0,Y 324.497,Z 774.597,A -85,B 0,C 180,E1 13306.911,E2 13306.911} C_VEL
LIN {X 0,Y 327.242,Z 779.396,A -85,B 0,C 180,E1 13304.766,E2 13304.766} C_VEL
LIN {X 0,Y 332.473,Z 788.601,A -85,B 0,C 180,E1 13301.366,E2 13301.366} C_VEL
LIN {X 0,Y 338.192,Z 799.163,A -85,B 0,C 180,E1 13298.266,E2 13298.266} C_VEL
LIN {X 0,Y 344.216,Z 810.673,A -85,B 0,C 180,E1 13295.457,E2 13295.457} C_VEL
LIN {X 0,Y 351.156,Z 824.933,A -85,B 0,C 180,E1 13292.6,E2 13292.6} C_VEL
LIN {X 0,Y 352.79,Z 828.966,A -85,B 0,C 180,E1 13291.953,E2 13291.953} C_VEL
LIN {X 0,Y 339.277,Z 1022.045,A -85,B 0,C 180,E1 13287.988,E2 13287.988} C_VEL
LIN {X 0,Y 336.286,Z 1044.379,A -85,B 0,C 180,E1 13287.347,E2 13287.347} C_VEL
LIN {X 0,Y 331.646,Z 1067.852,A -85,B 0,C 180,E1 13286.468,E2 13286.468} C_VEL
LIN {X 0,Y 326.423,Z 1088.321,A -85,B 0,C 180,E1 13285.481,E2 13285.481} C_VEL
LIN {X 0,Y 320.402,Z 1108.092,A -85,B 0,C 180,E1 13284.227,E2 13284.227} C_VEL
LIN {X 0,Y 313.117,Z 1129.229,A -85,B 0,C 180,E1 13282.513,E2 13282.513} C_VEL
LIN {X 0,Y 305.98,Z 1147.995,A -85,B 0,C 180,E1 13280.605,E2 13280.605} C_VEL
LIN {X 0,Y 298.249,Z 1166.672,A -85,B 0,C 180,E1 13278.236,E2 13278.236} C_VEL
LIN {X 0,Y 290.672,Z 1183.919,A -85,B 0,C 180,E1 13275.54,E2 13275.54} C_VEL
LIN {X 0,Y 283.228,Z 1200.419,A -85,B 0,C 180,E1 13272.396,E2 13272.396} C_VEL
LIN {X 0,Y 276.578,Z 1215.142,A -85,B 0,C 180,E1 13268.977,E2 13268.977} C_VEL
LIN {X 0,Y 270.64,Z 1228.56,A -85,B 0,C 180,E1 13265.191,E2 13265.191} C_VEL
LIN {X 0,Y 265.439,Z 1241.368,A -85,B 0,C 180,E1 13260.815,E2 13260.815} C_VEL
LIN {X 0,Y 261.647,Z 1252.182,A -85,B 0,C 180,E1 13256.313,E2 13256.313} C_VEL
LIN {X 0,Y 259.13,Z 1261.308,A -85,B 0,C 180,E1 13251.582,E2 13251.582} C_VEL
LIN {X 0,Y 257.829,Z 1268.859,A -85,B 0,C 180,E1 13246.676,E2 13246.676} C_VEL
LIN {X 0,Y 257.563,Z 1274.258,A -85,B 0,C 180,E1 13242.1,E2 13242.1} C_VEL
LIN {X 0,Y 257.864,Z 1277.938,A -85,B 0,C 180,E1 13237.575,E2 13237.575} C_VEL
LIN {X 0,Y 258.234,Z 1279.727,A -85,B 0,C 180,E1 13233.996,E2 13233.996} C_VEL
LIN {X 0,Y 258.427,Z 1280.491,A -85,B 0,C 180,E1 13230,E2 13230} C_VEL
LIN {X 0,Y 258.234,Z 1279.722,A -85,B 0,C 180,E1 13226.004,E2 13226.004} C_VEL
LIN {X 0,Y 257.864,Z 1277.929,A -85,B 0,C 180,E1 13222.425,E2 13222.425} C_VEL
LIN {X 0,Y 257.564,Z 1274.242,A -85,B 0,C 180,E1 13217.9,E2 13217.9} C_VEL
LIN {X 0,Y 257.83,Z 1268.845,A -85,B 0,C 180,E1 13213.324,E2 13213.324} C_VEL
LIN {X 0,Y 259.193,Z 1261.015,A -85,B 0,C 180,E1 13208.265,E2 13208.265} C_VEL
LIN {X 0,Y 261.647,Z 1252.148,A -85,B 0,C 180,E1 13203.687,E2 13203.687} C_VEL
LIN {X 0,Y 265.436,Z 1241.331,A -85,B 0,C 180,E1 13199.184,E2 13199.184} C_VEL
LIN {X 0,Y 270.346,Z 1229.208,A -85,B 0,C 180,E1 13195.023,E2 13195.023} C_VEL
LIN {X 0,Y 276.217,Z 1215.91,A -85,B 0,C 180,E1 13191.229,E2 13191.229} C_VEL
LIN {X 0,Y 282.802,Z 1201.251,A -85,B 0,C 180,E1 13187.799,E2 13187.799} C_VEL
LIN {X 0,Y 290.425,Z 1184.361,A -85,B 0,C 180,E1 13184.551,E2 13184.551} C_VEL
LIN {X 0,Y 297.978,Z 1167.188,A -85,B 0,C 180,E1 13181.85,E2 13181.85} C_VEL
LIN {X 0,Y 305.397,Z 1149.25,A -85,B 0,C 180,E1 13179.557,E2 13179.557} C_VEL
LIN {X 0,Y 312.798,Z 1129.896,A -85,B 0,C 180,E1 13177.561,E2 13177.561} C_VEL
LIN {X 0,Y 319.738,Z 1109.928,A -85,B 0,C 180,E1 13175.914,E2 13175.914} C_VEL
LIN {X 0,Y 326.102,Z 1089.098,A -85,B 0,C 180,E1 13174.576,E2 13174.576} C_VEL
LIN {X 0,Y 331.459,Z 1068.266,A -85,B 0,C 180,E1 13173.562,E2 13173.562} C_VEL
LIN {X 0,Y 336.015,Z 1045.475,A -85,B 0,C 180,E1 13172.699,E2 13172.699} C_VEL
LIN {X 0,Y 339.099,Z 1022.939,A -85,B 0,C 180,E1 13172.044,E2 13172.044} C_VEL
LIN {X 0,Y 346.854,Z 911.927,A -85,B 0,C 180,E1 13169.738,E2 13169.738} C_VEL
LIN {X 0,Y 352.6,Z 828.342,A -85,B 0,C 180,E1 13168.012,E2 13168.012} C_VEL
LIN {X 0,Y 345.892,Z 814.208,A -85,B 0,C 180,E1 13165.329,E2 13165.329} C_VEL
LIN {X 0,Y 339.277,Z 801.322,A -85,B 0,C 180,E1 13162.344,E2 13162.344} C_VEL
LIN {X 0,Y 334.11,Z 791.829,A -85,B 0,C 180,E1 13159.674,E2 13159.674} C_VEL
LIN {X 0,Y 330.255,Z 784.931,A -85,B 0,C 180,E1 13157.395,E2 13157.395} C_VEL
LIN {X 0,Y 325.937,Z 777.142,A -85,B 0,C 180,E1 13154.387,E2 13154.387} C_VEL
LIN {X 0,Y 322.94,Z 772.051,A -85,B 0,C 180,E1 13151.881,E2 13151.881} C_VEL
LIN {X 0,Y 320.801,Z 768.145,A -85,B 0,C 180,E1 13149.689,E2 13149.689} C_VEL
LIN {X 0,Y 318.612,Z 764.346,A -85,B 0,C 180,E1 13146.849,E2 13146.849} C_VEL
LIN {X 0,Y 315.759,Z 761.819,A -85,B 0,C 180,E1 13139.455,E2 13139.455} C_VEL
LIN {X 0,Y 316.171,Z 762.455,A -85,B 0,C 180,E1 13135.465,E2 13135.465} C_VEL
LIN {X 0,Y 318.937,Z 764.769,A -85,B 0,C 180,E1 13130.162,E2 13130.162} C_VEL
LIN {X 0,Y 321.331,Z 768.773,A -85,B 0,C 180,E1 13127.236,E2 13127.236} C_VEL
LIN {X 0,Y 323.194,Z 770.648,A -85,B 0,C 180,E1 13125.533,E2 13125.533} C_VEL
LIN {X 0,Y 326.361,Z 775.055,A -85,B 0,C 180,E1 13122.987,E2 13122.987} C_VEL
LIN {X 0,Y 331.249,Z 781.77,A -85,B 0,C 180,E1 13119.78,E2 13119.78} C_VEL
LIN {X 0,Y 335.47,Z 787.755,A -85,B 0,C 180,E1 13117.434,E2 13117.434} C_VEL
LIN {X 0,Y 340.498,Z 795.015,A -85,B 0,C 180,E1 13114.985,E2 13114.985} C_VEL
LIN {X 0,Y 348.384,Z 807.299,A -85,B 0,C 180,E1 13111.641,E2 13111.641} C_VEL
LIN {X 0,Y 352.53,Z 814.514,A -85,B 0,C 180,E1 13110.051,E2 13110.051} C_VEL
LIN {X 0,Y 343.015,Z 950.177,A -85,B 0,C 180,E1 13107.252,E2 13107.252} C_VEL
LIN {X 0,Y 341.015,Z 972.035,A -85,B 0,C 180,E1 13106.571,E2 13106.571} C_VEL
LIN {X 0,Y 337.852,Z 993.362,A -85,B 0,C 180,E1 13105.643,E2 13105.643} C_VEL
LIN {X 0,Y 333.646,Z 1014.405,A -85,B 0,C 180,E1 13104.453,E2 13104.453} C_VEL
LIN {X 0,Y 328.565,Z 1034.623,A -85,B 0,C 180,E1 13103.015,E2 13103.015} C_VEL
LIN {X 0,Y 323.017,Z 1052.938,A -85,B 0,C 180,E1 13101.403,E2 13101.403} C_VEL
LIN {X 0,Y 316.811,Z 1070.544,A -85,B 0,C 180,E1 13099.515,E2 13099.515} C_VEL
LIN {X 0,Y 310.09,Z 1087.523,A -85,B 0,C 180,E1 13097.319,E2 13097.319} C_VEL
LIN {X 0,Y 303.021,Z 1103.449,A -85,B 0,C 180,E1 13094.812,E2 13094.812} C_VEL
LIN {X 0,Y 295.792,Z 1118.349,A -85,B 0,C 180,E1 13091.955,E2 13091.955} C_VEL
LIN {X 0,Y 288.8,Z 1131.901,A -85,B 0,C 180,E1 13088.801,E2 13088.801} C_VEL
LIN {X 0,Y 282.081,Z 1144.203,A -85,B 0,C 180,E1 13085.292,E2 13085.292} C_VEL
LIN {X 0,Y 275.942,Z 1155.058,A -85,B 0,C 180,E1 13081.45,E2 13081.45} C_VEL
LIN {X 0,Y 270.32,Z 1164.988,A -85,B 0,C 180,E1 13077.061,E2 13077.061} C_VEL
LIN {X 0,Y 266.098,Z 1172.684,A -85,B 0,C 180,E1 13072.769,E2 13072.769} C_VEL
LIN {X 0,Y 262.815,Z 1178.916,A -85,B 0,C 180,E1 13068.177,E2 13068.177} C_VEL
LIN {X 0,Y 260.505,Z 1183.788,A -85,B 0,C 180,E1 13063.314,E2 13063.314} C_VEL
LIN {X 0,Y 259.242,Z 1187,A -85,B 0,C 180,E1 13058.651,E2 13058.651} C_VEL
LIN {X 0,Y 258.612,Z 1188.723,A -85,B 0,C 180,E1 13053.99,E2 13053.99} C_VEL
LIN {X 0,Y 258.487,Z 1189.197,A -85,B 0,C 180,E1 13049.113,E2 13049.113} C_VEL
LIN {X 0,Y 258.734,Z 1188.409,A -85,B 0,C 180,E1 13044.679,E2 13044.679} C_VEL
LIN {X 0,Y 259.57,Z 1186.113,A -85,B 0,C 180,E1 13039.794,E2 13039.794} C_VEL
LIN {X 0,Y 261.091,Z 1182.568,A -85,B 0,C 180,E1 13035.133,E2 13035.133} C_VEL
LIN {X 0,Y 263.591,Z 1177.441,A -85,B 0,C 180,E1 13030.501,E2 13030.501} C_VEL
LIN {X 0,Y 267.175,Z 1170.682,A -85,B 0,C 180,E1 13025.927,E2 13025.927} C_VEL
LIN {X 0,Y 271.903,Z 1162.281,A -85,B 0,C 180,E1 13021.507,E2 13021.507} C_VEL
LIN {X 0,Y 277.682,Z 1152.155,A -85,B 0,C 180,E1 13017.31,E2 13017.31} C_VEL
LIN {X 0,Y 283.742,Z 1141.261,A -85,B 0,C 180,E1 13013.702,E2 13013.702} C_VEL
LIN {X 0,Y 290.677,Z 1128.445,A -85,B 0,C 180,E1 13010.225,E2 13010.225} C_VEL
LIN {X 0,Y 298,Z 1114.198,A -85,B 0,C 180,E1 13007.071,E2 13007.071} C_VEL
LIN {X 0,Y 305.233,Z 1098.776,A -85,B 0,C 180,E1 13004.297,E2 13004.297} C_VEL
LIN {X 0,Y 312.484,Z 1081.849,A -85,B 0,C 180,E1 13001.797,E2 13001.797} C_VEL
LIN {X 0,Y 319.07,Z 1064.735,A -85,B 0,C 180,E1 12999.71,E2 12999.71} C_VEL
LIN {X 0,Y 325.07,Z 1046.766,A -85,B 0,C 180,E1 12997.915,E2 12997.915} C_VEL
LIN {X 0,Y 330.635,Z 1027.212,A -85,B 0,C 180,E1 12996.319,E2 12996.319} C_VEL
LIN {X 0,Y 335.351,Z 1007.184,A -85,B 0,C 180,E1 12995,E2 12995} C_VEL
LIN {X 0,Y 339.095,Z 986.501,A -85,B 0,C 180,E1 12993.929,E2 12993.929} C_VEL
LIN {X 0,Y 340.854,Z 974.003,A -85,B 0,C 180,E1 12993.407,E2 12993.407} C_VEL
LIN {X 0,Y 341.206,Z 966.657,A -85,B 0,C 180,E1 12992.984,E2 12992.984} C_VEL
LIN {X 0,Y 339.677,Z 948.416,A -85,B 0,C 180,E1 12991.586,E2 12991.586} C_VEL
LIN {X 0,Y 339.658,Z 940.915,A -85,B 0,C 180,E1 12991.265,E2 12991.265} C_VEL
LIN {X 0,Y 348.533,Z 818.695,A -85,B 0,C 180,E1 12988.766,E2 12988.766} C_VEL
LIN {X 0,Y 342.248,Z 808.35,A -85,B 0,C 180,E1 12986.177,E2 12986.177} C_VEL
LIN {X 0,Y 336.206,Z 798.933,A -85,B 0,C 180,E1 12983.346,E2 12983.346} C_VEL
LIN {X 0,Y 331.255,Z 791.726,A -85,B 0,C 180,E1 12980.681,E2 12980.681} C_VEL
LIN {X 0,Y 328.123,Z 787.255,A -85,B 0,C 180,E1 12978.753,E2 12978.753} C_VEL
LIN {X 0,Y 324.853,Z 782.645,A -85,B 0,C 180,E1 12976.449,E2 12976.449} C_VEL
LIN {X 0,Y 321.393,Z 777.734,A -85,B 0,C 180,E1 12973.493,E2 12973.493} C_VEL
LIN {X 0,Y 318.423,Z 774.015,A -85,B 0,C 180,E1 12970.219,E2 12970.219} C_VEL
LIN {X 0,Y 317.676,Z 772.33,A -85,B 0,C 180,E1 12969.055,E2 12969.055} C_VEL
LIN {X 0,Y 315.008,Z 770.042,A -85,B 0,C 180,E1 12961.819,E2 12961.819} C_VEL
LIN {X 0,Y 315.576,Z 770.81,A -85,B 0,C 180,E1 12957.458,E2 12957.458} C_VEL
LIN {X 0,Y 317.835,Z 772.6,A -85,B 0,C 180,E1 12953.135,E2 12953.135} C_VEL
LIN {X 0,Y 320.31,Z 777.17,A -85,B 0,C 180,E1 12949.933,E2 12949.933} C_VEL
LIN {X 0,Y 323.082,Z 782.335,A -85,B 0,C 180,E1 12947.216,E2 12947.216} C_VEL
LIN {X 0,Y 325.758,Z 787.18,A -85,B 0,C 180,E1 12945.059,E2 12945.059} C_VEL
LIN {X 0,Y 331.09,Z 796.846,A -85,B 0,C 180,E1 12941.513,E2 12941.513} C_VEL
LIN {X 0,Y 336.571,Z 807.414,A -85,B 0,C 180,E1 12938.477,E2 12938.477} C_VEL
LIN {X 0,Y 342.419,Z 819.007,A -85,B 0,C 180,E1 12935.688,E2 12935.688} C_VEL
LIN {X 0,Y 348.68,Z 832.487,A -85,B 0,C 180,E1 12933.031,E2 12933.031} C_VEL
LIN {X 0,Y 335.047,Z 1020.633,A -85,B 0,C 180,E1 12929.164,E2 12929.164} C_VEL
LIN {X 0,Y 331.979,Z 1042.959,A -85,B 0,C 180,E1 12928.526,E2 12928.526} C_VEL
LIN {X 0,Y 327.238,Z 1066.431,A -85,B 0,C 180,E1 12927.651,E2 12927.651} C_VEL
LIN {X 0,Y 321.686,Z 1087.539,A -85,B 0,C 180,E1 12926.637,E2 12926.637} C_VEL
LIN {X 0,Y 315.355,Z 1107.682,A -85,B 0,C 180,E1 12925.36,E2 12925.36} C_VEL
LIN {X 0,Y 308.192,Z 1127.738,A -85,B 0,C 180,E1 12923.732,E2 12923.732} C_VEL
LIN {X 0,Y 300.653,Z 1146.848,A -85,B 0,C 180,E1 12921.789,E2 12921.789} C_VEL
LIN {X 0,Y 292.76,Z 1165.197,A -85,B 0,C 180,E1 12919.455,E2 12919.455} C_VEL
LIN {X 0,Y 285.11,Z 1181.905,A -85,B 0,C 180,E1 12916.838,E2 12916.838} C_VEL
LIN {X 0,Y 277.523,Z 1198.033,A -85,B 0,C 180,E1 12913.766,E2 12913.766} C_VEL
LIN {X 0,Y 270.436,Z 1212.821,A -85,B 0,C 180,E1 12910.315,E2 12910.315} C_VEL
LIN {X 0,Y 264.098,Z 1226.375,A -85,B 0,C 180,E1 12906.468,E2 12906.468} C_VEL
LIN {X 0,Y 258.646,Z 1238.913,A -85,B 0,C 180,E1 12902.157,E2 12902.157} C_VEL
LIN {X 0,Y 254.321,Z 1250.186,A -85,B 0,C 180,E1 12897.385,E2 12897.385} C_VEL
LIN {X 0,Y 251.467,Z 1259.567,A -85,B 0,C 180,E1 12892.439,E2 12892.439} C_VEL
LIN {X 0,Y 249.948,Z 1267.406,A -85,B 0,C 180,E1 12887.218,E2 12887.218} C_VEL
LIN {X 0,Y 249.614,Z 1272.577,A -85,B 0,C 180,E1 12882.727,E2 12882.727} C_VEL
LIN {X 0,Y 249.907,Z 1276.384,A -85,B 0,C 180,E1 12878.049,E2 12878.049} C_VEL
LIN {X 0,Y 250.319,Z 1278.246,A -85,B 0,C 180,E1 12874.352,E2 12874.352} C_VEL
LIN {X 0,Y 250.535,Z 1279.059,A -85,B 0,C 180,E1 12870.457,E2 12870.457} C_VEL
LIN {X 0,Y 250.385,Z 1278.573,A -85,B 0,C 180,E1 12866.566,E2 12866.566} C_VEL
LIN {X 0,Y 249.98,Z 1276.799,A -85,B 0,C 180,E1 12862.647,E2 12862.647} C_VEL
LIN {X 0,Y 249.655,Z 1273.677,A -85,B 0,C 180,E1 12858.449,E2 12858.449} C_VEL
LIN {X 0,Y 249.841,Z 1268.293,A -85,B 0,C 180,E1 12853.493,E2 12853.493} C_VEL
LIN {X 0,Y 251.082,Z 1261.168,A -85,B 0,C 180,E1 12848.509,E2 12848.509} C_VEL
LIN {X 0,Y 253.499,Z 1252.547,A -85,B 0,C 180,E1 12843.785,E2 12843.785} C_VEL
LIN {X 0,Y 257.291,Z 1242.135,A -85,B 0,C 180,E1 12839.14,E2 12839.14} C_VEL
LIN {X 0,Y 262.256,Z 1230.497,A -85,B 0,C 180,E1 12834.853,E2 12834.853} C_VEL
LIN {X 0,Y 268.564,Z 1216.738,A -85,B 0,C 180,E1 12830.737,E2 12830.737} C_VEL
LIN {X 0,Y 275.748,Z 1201.572,A -85,B 0,C 180,E1 12827.026,E2 12827.026} C_VEL
LIN {X 0,Y 283.615,Z 1185.023,A -85,B 0,C 180,E1 12823.723,E2 12823.723} C_VEL
LIN {X 0,Y 291.388,Z 1168.175,A -85,B 0,C 180,E1 12820.985,E2 12820.985} C_VEL
LIN {X 0,Y 299.295,Z 1149.867,A -85,B 0,C 180,E1 12818.583,E2 12818.583} C_VEL
LIN {X 0,Y 307.212,Z 1130.111,A -85,B 0,C 180,E1 12816.499,E2 12816.499} C_VEL
LIN {X 0,Y 314.34,Z 1110.531,A -85,B 0,C 180,E1 12814.853,E2 12814.853} C_VEL
LIN {X 0,Y 320.813,Z 1090.073,A -85,B 0,C 180,E1 12813.522,E2 12813.522} C_VEL
LIN {X 0,Y 326.646,Z 1068.491,A -85,B 0,C 180,E1 12812.449,E2 12812.449} C_VEL
LIN {X 0,Y 331.273,Z 1046.66,A -85,B 0,C 180,E1 12811.604,E2 12811.604} C_VEL
LIN {X 0,Y 334.527,Z 1024.326,A -85,B 0,C 180,E1 12810.942,E2 12810.942} C_VEL
LIN {X 0,Y 337.321,Z 989.531,A -85,B 0,C 180,E1 12810.182,E2 12810.182} C_VEL
LIN {X 0,Y 348.508,Z 832.24,A -85,B 0,C 180,E1 12806.955,E2 12806.955} C_VEL
LIN {X 0,Y 341.855,Z 817.988,A -85,B 0,C 180,E1 12804.125,E2 12804.125} C_VEL
LIN {X 0,Y 335.799,Z 806.078,A -85,B 0,C 180,E1 12801.209,E2 12801.209} C_VEL
LIN {X 0,Y 330.205,Z 795.389,A -85,B 0,C 180,E1 12798.055,E2 12798.055} C_VEL
LIN {X 0,Y 324.6,Z 785.004,A -85,B 0,C 180,E1 12794.175,E2 12794.175} C_VEL
LIN {X 0,Y 321.29,Z 779.289,A -85,B 0,C 180,E1 12791.306,E2 12791.306} C_VEL
LIN {X 0,Y 319.495,Z 775.838,A -85,B 0,C 180,E1 12789.365,E2 12789.365} C_VEL
LIN {X 0,Y 317.51,Z 772.236,A -85,B 0,C 180,E1 12786.691,E2 12786.691} C_VEL
LIN {X 0,Y 314.784,Z 769.761,A -85,B 0,C 180,E1 12779.454,E2 12779.454} C_VEL
LIN {X 0,Y 315.149,Z 770.352,A -85,B 0,C 180,E1 12775.633,E2 12775.633} C_VEL
LIN {X 0,Y 317.766,Z 772.623,A -85,B 0,C 180,E1 12770.4,E2 12770.4} C_VEL
LIN {X 0,Y 320.187,Z 776.669,A -85,B 0,C 180,E1 12767.373,E2 12767.373} C_VEL
LIN {X 0,Y 321.867,Z 778.474,A -85,B 0,C 180,E1 12765.794,E2 12765.794} C_VEL
LIN {X 0,Y 325.16,Z 782.981,A -85,B 0,C 180,E1 12763.107,E2 12763.107} C_VEL
LIN {X 0,Y 329.703,Z 789.58,A -85,B 0,C 180,E1 12760.052,E2 12760.052} C_VEL
LIN {X 0,Y 333.782,Z 795.469,A -85,B 0,C 180,E1 12757.732,E2 12757.732} C_VEL
LIN {X 0,Y 338.805,Z 803.018,A -85,B 0,C 180,E1 12755.224,E2 12755.224} C_VEL
LIN {X 0,Y 345.83,Z 814.208,A -85,B 0,C 180,E1 12752.165,E2 12752.165} C_VEL
LIN {X 0,Y 348.424,Z 818.9,A -85,B 0,C 180,E1 12751.119,E2 12751.119} C_VEL
LIN {X 0,Y 338.855,Z 950.961,A -85,B 0,C 180,E1 12748.393,E2 12748.393} C_VEL
LIN {X 0,Y 336.792,Z 972.996,A -85,B 0,C 180,E1 12747.708,E2 12747.708} C_VEL
LIN {X 0,Y 333.545,Z 994.308,A -85,B 0,C 180,E1 12746.783,E2 12746.783} C_VEL
LIN {X 0,Y 329.296,Z 1015.091,A -85,B 0,C 180,E1 12745.614,E2 12745.614} C_VEL
LIN {X 0,Y 324.179,Z 1035.049,A -85,B 0,C 180,E1 12744.207,E2 12744.207} C_VEL
LIN {X 0,Y 318.158,Z 1054.334,A -85,B 0,C 180,E1 12742.513,E2 12742.513} C_VEL
LIN {X 0,Y 311.745,Z 1071.941,A -85,B 0,C 180,E1 12740.618,E2 12740.618} C_VEL
LIN {X 0,Y 304.79,Z 1088.921,A -85,B 0,C 180,E1 12738.411,E2 12738.411} C_VEL
LIN {X 0,Y 297.586,Z 1104.577,A -85,B 0,C 180,E1 12735.933,E2 12735.933} C_VEL
LIN {X 0,Y 290.043,Z 1119.565,A -85,B 0,C 180,E1 12733.042,E2 12733.042} C_VEL
LIN {X 0,Y 282.654,Z 1133.305,A -85,B 0,C 180,E1 12729.81,E2 12729.81} C_VEL
LIN {X 0,Y 275.63,Z 1145.608,A -85,B 0,C 180,E1 12726.247,E2 12726.247} C_VEL
LIN {X 0,Y 269.182,Z 1156.465,A -85,B 0,C 180,E1 12722.335,E2 12722.335} C_VEL
LIN {X 0,Y 263.247,Z 1166.396,A -85,B 0,C 180,E1 12717.85,E2 12717.85} C_VEL
LIN {X 0,Y 258.772,Z 1174.091,A -85,B 0,C 180,E1 12713.451,E2 12713.451} C_VEL
LIN {X 0,Y 255.275,Z 1180.319,A -85,B 0,C 180,E1 12708.734,E2 12708.734} C_VEL
LIN {X 0,Y 252.792,Z 1185.188,A -85,B 0,C 180,E1 12703.728,E2 12703.728} C_VEL
LIN {X 0,Y 251.43,Z 1188.396,A -85,B 0,C 180,E1 12698.922,E2 12698.922} C_VEL
LIN {X 0,Y 250.747,Z 1190.114,A -85,B 0,C 180,E1 12694.116,E2 12694.116} C_VEL
LIN {X 0,Y 250.609,Z 1190.587,A -85,B 0,C 180,E1 12689.086,E2 12689.086} C_VEL
LIN {X 0,Y 250.877,Z 1189.802,A -85,B 0,C 180,E1 12684.511,E2 12684.511} C_VEL
LIN {X 0,Y 251.782,Z 1187.51,A -85,B 0,C 180,E1 12679.475,E2 12679.475} C_VEL
LIN {X 0,Y 253.42,Z 1183.969,A -85,B 0,C 180,E1 12674.672,E2 12674.672} C_VEL
LIN {X 0,Y 256.1,Z 1178.845,A -85,B 0,C 180,E1 12669.906,E2 12669.906} C_VEL
LIN {X 0,Y 259.932,Z 1172.074,A -85,B 0,C 180,E1 12665.204,E2 12665.204} C_VEL
LIN {X 0,Y 264.731,Z 1164.031,A -85,B 0,C 180,E1 12660.843,E2 12660.843} C_VEL
LIN {X 0,Y 270.723,Z 1154.023,A -85,B 0,C 180,E1 12656.584,E2 12656.584} C_VEL
LIN {X 0,Y 277.371,Z 1142.662,A -85,B 0,C 180,E1 12652.729,E2 12652.729} C_VEL
LIN {X 0,Y 284.62,Z 1129.843,A -85,B 0,C 180,E1 12649.202,E2 12649.202} C_VEL
LIN {X 0,Y 292.247,Z 1115.594,A -85,B 0,C 180,E1 12646.013,E2 12646.013} C_VEL
LIN {X 0,Y 299.761,Z 1100.169,A -85,B 0,C 180,E1 12643.215,E2 12643.215} C_VEL
LIN {X 0,Y 307.275,Z 1083.238,A -85,B 0,C 180,E1 12640.699,E2 12640.699} C_VEL
LIN {X 0,Y 314.074,Z 1066.162,A -85,B 0,C 180,E1 12638.607,E2 12638.607} C_VEL
LIN {X 0,Y 320.257,Z 1048.238,A -85,B 0,C 180,E1 12636.81,E2 12636.81} C_VEL
LIN {X 0,Y 325.99,Z 1028.743,A -85,B 0,C 180,E1 12635.214,E2 12635.214} C_VEL
LIN {X 0,Y 330.751,Z 1009.285,A -85,B 0,C 180,E1 12633.923,E2 12633.923} C_VEL
LIN {X 0,Y 334.646,Z 988.517,A -85,B 0,C 180,E1 12632.839,E2 12632.839} C_VEL
LIN {X 0,Y 337.536,Z 967.107,A -85,B 0,C 180,E1 12631.99,E2 12631.99} C_VEL
LIN {X 0,Y 339.453,Z 944.109,A -85,B 0,C 180,E1 12631.337,E2 12631.337} C_VEL
LIN {X 0,Y 339.658,Z 940.915,A -85,B 0,C 180,E1 12631.265,E2 12631.265} C_VEL
LIN {X 0,Y 339.658,Z 933.372,A -85,B 0,C 180,E1 12630.952,E2 12630.952} C_VEL
LIN {X 0,Y 338.031,Z 913.726,A -85,B 0,C 180,E1 12629.617,E2 12629.617} C_VEL
LIN {X 0,Y 338.164,Z 907.234,A -85,B 0,C 180,E1 12629.374,E2 12629.374} C_VEL
LIN {X 0,Y 344.536,Z 823.111,A -85,B 0,C 180,E1 12627.667,E2 12627.667} C_VEL
LIN {X 0,Y 337.928,Z 812.122,A -85,B 0,C 180,E1 12624.751,E2 12624.751} C_VEL
LIN {X 0,Y 332.323,Z 803.397,A -85,B 0,C 180,E1 12621.906,E2 12621.906} C_VEL
LIN {X 0,Y 328.521,Z 797.818,A -85,B 0,C 180,E1 12619.699,E2 12619.699} C_VEL
LIN {X 0,Y 326.241,Z 794.488,A -85,B 0,C 180,E1 12618.217,E2 12618.217} C_VEL
LIN {X 0,Y 323.312,Z 790.219,A -85,B 0,C 180,E1 12616.069,E2 12616.069} C_VEL
LIN {X 0,Y 320.049,Z 785.466,A -85,B 0,C 180,E1 12613.183,E2 12613.183} C_VEL
LIN {X 0,Y 317.127,Z 781.577,A -85,B 0,C 180,E1 12609.803,E2 12609.803} C_VEL
LIN {X 0,Y 316.458,Z 780.166,A -85,B 0,C 180,E1 12608.723,E2 12608.723} C_VEL
LIN {X 0,Y 314.026,Z 777.968,A -85,B 0,C 180,E1 12601.642,E2 12601.642} C_VEL
LIN {X 0,Y 314.721,Z 778.902,A -85,B 0,C 180,E1 12597.087,E2 12597.087} C_VEL
LIN {X 0,Y 316.672,Z 780.431,A -85,B 0,C 180,E1 12593.383,E2 12593.383} C_VEL
LIN {X 0,Y 318.991,Z 784.883,A -85,B 0,C 180,E1 12590.256,E2 12590.256} C_VEL
LIN {X 0,Y 321.677,Z 790.068,A -85,B 0,C 180,E1 12587.525,E2 12587.525} C_VEL
LIN {X 0,Y 324.339,Z 795.06,A -85,B 0,C 180,E1 12585.312,E2 12585.312} C_VEL
LIN {X 0,Y 329.09,Z 804.002,A -85,B 0,C 180,E1 12582.039,E2 12582.039} C_VEL
LIN {X 0,Y 334.257,Z 814.281,A -85,B 0,C 180,E1 12579.056,E2 12579.056} C_VEL
LIN {X 0,Y 339.849,Z 825.758,A -85,B 0,C 180,E1 12576.277,E2 12576.277} C_VEL
LIN {X 0,Y 344.657,Z 836.519,A -85,B 0,C 180,E1 12574.124,E2 12574.124} C_VEL
LIN {X 0,Y 330.963,Z 1019.222,A -85,B 0,C 180,E1 12570.37,E2 12570.37} C_VEL
LIN {X 0,Y 327.807,Z 1041.606,A -85,B 0,C 180,E1 12569.733,E2 12569.733} C_VEL
LIN {X 0,Y 323.017,Z 1064.823,A -85,B 0,C 180,E1 12568.874,E2 12568.874} C_VEL
LIN {X 0,Y 317.492,Z 1085.465,A -85,B 0,C 180,E1 12567.9,E2 12567.9} C_VEL
LIN {X 0,Y 311.062,Z 1105.414,A -85,B 0,C 180,E1 12566.657,E2 12566.657} C_VEL
LIN {X 0,Y 303.67,Z 1125.601,A -85,B 0,C 180,E1 12565.047,E2 12565.047} C_VEL
LIN {X 0,Y 296.055,Z 1144.385,A -85,B 0,C 180,E1 12563.167,E2 12563.167} C_VEL
LIN {X 0,Y 287.694,Z 1163.099,A -85,B 0,C 180,E1 12560.805,E2 12560.805} C_VEL
LIN {X 0,Y 279.441,Z 1180.428,A -85,B 0,C 180,E1 12558.092,E2 12558.092} C_VEL
LIN {X 0,Y 271.513,Z 1196.552,A -85,B 0,C 180,E1 12554.993,E2 12554.993} C_VEL
LIN {X 0,Y 263.808,Z 1211.837,A -85,B 0,C 180,E1 12551.372,E2 12551.372} C_VEL
LIN {X 0,Y 257.018,Z 1225.582,A -85,B 0,C 180,E1 12547.363,E2 12547.363} C_VEL
LIN {X 0,Y 251.098,Z 1238.394,A -85,B 0,C 180,E1 12542.788,E2 12542.788} C_VEL
LIN {X 0,Y 246.574,Z 1249.571,A -85,B 0,C 180,E1 12537.874,E2 12537.874} C_VEL
LIN {X 0,Y 243.555,Z 1258.909,A -85,B 0,C 180,E1 12532.699,E2 12532.699} C_VEL
LIN {X 0,Y 242.033,Z 1266.252,A -85,B 0,C 180,E1 12527.551,E2 12527.551} C_VEL
LIN {X 0,Y 241.675,Z 1271.634,A -85,B 0,C 180,E1 12522.666,E2 12522.666} C_VEL
LIN {X 0,Y 241.993,Z 1275.112,A -85,B 0,C 180,E1 12518.075,E2 12518.075} C_VEL
LIN {X 0,Y 242.436,Z 1276.932,A -85,B 0,C 180,E1 12514.257,E2 12514.257} C_VEL
LIN {X 0,Y 242.661,Z 1277.693,A -85,B 0,C 180,E1 12510.236,E2 12510.236} C_VEL
LIN {X 0,Y 242.472,Z 1277.094,A -85,B 0,C 180,E1 12506.217,E2 12506.217} C_VEL
LIN {X 0,Y 242.046,Z 1275.387,A -85,B 0,C 180,E1 12502.404,E2 12502.404} C_VEL
LIN {X 0,Y 241.705,Z 1272.244,A -85,B 0,C 180,E1 12498.063,E2 12498.063} C_VEL
LIN {X 0,Y 241.963,Z 1266.84,A -85,B 0,C 180,E1 12492.939,E2 12492.939} C_VEL
LIN {X 0,Y 243.35,Z 1259.697,A -85,B 0,C 180,E1 12487.791,E2 12487.791} C_VEL
LIN {X 0,Y 246.028,Z 1250.975,A -85,B 0,C 180,E1 12482.874,E2 12482.874} C_VEL
LIN {X 0,Y 250.336,Z 1240.071,A -85,B 0,C 180,E1 12477.914,E2 12477.914} C_VEL
LIN {X 0,Y 255.701,Z 1228.307,A -85,B 0,C 180,E1 12473.534,E2 12473.534} C_VEL
LIN {X 0,Y 262.464,Z 1214.483,A -85,B 0,C 180,E1 12469.352,E2 12469.352} C_VEL
LIN {X 0,Y 269.65,Z 1200.084,A -85,B 0,C 180,E1 12465.807,E2 12465.807} C_VEL
LIN {X 0,Y 277.884,Z 1183.54,A -85,B 0,C 180,E1 12462.473,E2 12462.473} C_VEL
LIN {X 0,Y 285.984,Z 1166.699,A -85,B 0,C 180,E1 12459.723,E2 12459.723} C_VEL
LIN {X 0,Y 294.19,Z 1148.398,A -85,B 0,C 180,E1 12457.32,E2 12457.32} C_VEL
LIN {X 0,Y 302.387,Z 1128.653,A -85,B 0,C 180,E1 12455.245,E2 12455.245} C_VEL
LIN {X 0,Y 309.738,Z 1109.081,A -85,B 0,C 180,E1 12453.611,E2 12453.611} C_VEL
LIN {X 0,Y 316.033,Z 1089.781,A -85,B 0,C 180,E1 12452.36,E2 12452.36} C_VEL
LIN {X 0,Y 322.226,Z 1067.637,A -85,B 0,C 180,E1 12451.258,E2 12451.258} C_VEL
LIN {X 0,Y 326.993,Z 1045.82,A -85,B 0,C 180,E1 12450.413,E2 12450.413} C_VEL
LIN {X 0,Y 330.362,Z 1023.386,A -85,B 0,C 180,E1 12449.749,E2 12449.749} C_VEL
LIN {X 0,Y 333.137,Z 990.522,A -85,B 0,C 180,E1 12449.027,E2 12449.027} C_VEL
LIN {X 0,Y 344.49,Z 836.155,A -85,B 0,C 180,E1 12445.859,E2 12445.859} C_VEL
LIN {X 0,Y 338.2,Z 822.472,A -85,B 0,C 180,E1 12443.015,E2 12443.015} C_VEL
LIN {X 0,Y 332.092,Z 810.063,A -85,B 0,C 180,E1 12439.844,E2 12439.844} C_VEL
LIN {X 0,Y 327.035,Z 800.301,A -85,B 0,C 180,E1 12436.747,E2 12436.747} C_VEL
LIN {X 0,Y 322.61,Z 791.877,A -85,B 0,C 180,E1 12433.441,E2 12433.441} C_VEL
LIN {X 0,Y 319.846,Z 786.827,A -85,B 0,C 180,E1 12430.901,E2 12430.901} C_VEL
LIN {X 0,Y 318.123,Z 783.423,A -85,B 0,C 180,E1 12428.95,E2 12428.95} C_VEL
LIN {X 0,Y 316.284,Z 780.063,A -85,B 0,C 180,E1 12426.352,E2 12426.352} C_VEL
LIN {X 0,Y 313.801,Z 777.68,A -85,B 0,C 180,E1 12419.269,E2 12419.269} C_VEL
LIN {X 0,Y 314.275,Z 778.432,A -85,B 0,C 180,E1 12415.255,E2 12415.255} C_VEL
LIN {X 0,Y 316.601,Z 780.471,A -85,B 0,C 180,E1 12410.639,E2 12410.639} C_VEL
LIN {X 0,Y 319.045,Z 784.564,A -85,B 0,C 180,E1 12407.511,E2 12407.511} C_VEL
LIN {X 0,Y 320.503,Z 786.204,A -85,B 0,C 180,E1 12406.101,E2 12406.101} C_VEL
LIN {X 0,Y 324.39,Z 791.844,A -85,B 0,C 180,E1 12402.881,E2 12402.881} C_VEL
LIN {X 0,Y 328.033,Z 797.164,A -85,B 0,C 180,E1 12400.41,E2 12400.41} C_VEL
LIN {X 0,Y 333.112,Z 804.542,A -85,B 0,C 180,E1 12397.499,E2 12397.499} C_VEL
LIN {X 0,Y 339.606,Z 815.012,A -85,B 0,C 180,E1 12394.308,E2 12394.308} C_VEL
LIN {X 0,Y 344.454,Z 823.106,A -85,B 0,C 180,E1 12392.216,E2 12392.216} C_VEL
LIN {X 0,Y 334.832,Z 951.746,A -85,B 0,C 180,E1 12389.562,E2 12389.562} C_VEL
LIN {X 0,Y 332.726,Z 973.702,A -85,B 0,C 180,E1 12388.882,E2 12388.882} C_VEL
LIN {X 0,Y 329.422,Z 994.97,A -85,B 0,C 180,E1 12387.967,E2 12387.967} C_VEL
LIN {X 0,Y 325.034,Z 1015.987,A -85,B 0,C 180,E1 12386.792,E2 12386.792} C_VEL
LIN {X 0,Y 319.937,Z 1035.472,A -85,B 0,C 180,E1 12385.432,E2 12385.432} C_VEL
LIN {X 0,Y 313.712,Z 1054.866,A -85,B 0,C 180,E1 12383.739,E2 12383.739} C_VEL
LIN {X 0,Y 306.798,Z 1073.338,A -85,B 0,C 180,E1 12381.757,E2 12381.757} C_VEL
LIN {X 0,Y 299.604,Z 1090.319,A -85,B 0,C 180,E1 12379.541,E2 12379.541} C_VEL
LIN {X 0,Y 291.956,Z 1106.354,A -85,B 0,C 180,E1 12376.983,E2 12376.983} C_VEL
LIN {X 0,Y 284.302,Z 1120.967,A -85,B 0,C 180,E1 12374.133,E2 12374.133} C_VEL
LIN {X 0,Y 276.599,Z 1134.709,A -85,B 0,C 180,E1 12370.864,E2 12370.864} C_VEL
LIN {X 0,Y 269.26,Z 1147.013,A -85,B 0,C 180,E1 12367.247,E2 12367.247} C_VEL
LIN {X 0,Y 262.491,Z 1157.872,A -85,B 0,C 180,E1 12363.264,E2 12363.264} C_VEL
LIN {X 0,Y 256.229,Z 1167.804,A -85,B 0,C 180,E1 12358.683,E2 12358.683} C_VEL
LIN {X 0,Y 251.487,Z 1175.497,A -85,B 0,C 180,E1 12354.173,E2 12354.173} C_VEL
LIN {X 0,Y 247.61,Z 1181.993,A -85,B 0,C 180,E1 12349.091,E2 12349.091} C_VEL
LIN {X 0,Y 245,Z 1186.768,A -85,B 0,C 180,E1 12343.932,E2 12343.932} C_VEL
LIN {X 0,Y 243.567,Z 1189.889,A -85,B 0,C 180,E1 12338.974,E2 12338.974} C_VEL
LIN {X 0,Y 242.864,Z 1191.565,A -85,B 0,C 180,E1 12334.013,E2 12334.013} C_VEL
LIN {X 0,Y 242.731,Z 1191.978,A -85,B 0,C 180,E1 12329.056,E2 12329.056} C_VEL
LIN {X 0,Y 243.022,Z 1191.194,A -85,B 0,C 180,E1 12324.333,E2 12324.333} C_VEL
LIN {X 0,Y 244.001,Z 1188.906,A -85,B 0,C 180,E1 12319.135,E2 12319.135} C_VEL
LIN {X 0,Y 245.872,Z 1185.146,A -85,B 0,C 180,E1 12313.947,E2 12313.947} C_VEL
LIN {X 0,Y 248.807,Z 1179.981,A -85,B 0,C 180,E1 12309.044,E2 12309.044} C_VEL
LIN {X 0,Y 252.94,Z 1173.126,A -85,B 0,C 180,E1 12304.227,E2 12304.227} C_VEL
LIN {X 0,Y 258.369,Z 1164.496,A -85,B 0,C 180,E1 12299.54,E2 12299.54} C_VEL
LIN {X 0,Y 264.768,Z 1154.42,A -85,B 0,C 180,E1 12295.235,E2 12295.235} C_VEL
LIN {X 0,Y 271.885,Z 1142.763,A -85,B 0,C 180,E1 12291.306,E2 12291.306} C_VEL
LIN {X 0,Y 279.551,Z 1129.657,A -85,B 0,C 180,E1 12287.748,E2 12287.748} C_VEL
LIN {X 0,Y 287.157,Z 1115.889,A -85,B 0,C 180,E1 12284.697,E2 12284.697} C_VEL
LIN {X 0,Y 294.661,Z 1101.036,A -85,B 0,C 180,E1 12282.004,E2 12282.004} C_VEL
LIN {X 0,Y 302.182,Z 1084.629,A -85,B 0,C 180,E1 12279.563,E2 12279.563} C_VEL
LIN {X 0,Y 309.377,Z 1067.097,A -85,B 0,C 180,E1 12277.416,E2 12277.416} C_VEL
LIN {X 0,Y 315.927,Z 1048.669,A -85,B 0,C 180,E1 12275.577,E2 12275.577} C_VEL
LIN {X 0,Y 321.693,Z 1029.469,A -85,B 0,C 180,E1 12274.019,E2 12274.019} C_VEL
LIN {X 0,Y 326.715,Z 1009.226,A -85,B 0,C 180,E1 12272.694,E2 12272.694} C_VEL
LIN {X 0,Y 330.686,Z 988.52,A -85,B 0,C 180,E1 12271.626,E2 12271.626} C_VEL
LIN {X 0,Y 333.537,Z 967.448,A -85,B 0,C 180,E1 12270.805,E2 12270.805} C_VEL
LIN {X 0,Y 335.632,Z 942.092,A -85,B 0,C 180,E1 12270.105,E2 12270.105} C_VEL
LIN {X 0,Y 338.164,Z 907.234,A -85,B 0,C 180,E1 12269.374,E2 12269.374} C_VEL
LIN {X 0,Y 338.265,Z 899.674,A -85,B 0,C 180,E1 12269.071,E2 12269.071} C_VEL
LIN {X 0,Y 336.908,Z 879.999,A -85,B 0,C 180,E1 12267.726,E2 12267.726} C_VEL
LIN {X 0,Y 337.096,Z 873.497,A -85,B 0,C 180,E1 12267.485,E2 12267.485} C_VEL
LIN {X 0,Y 340.662,Z 827.595,A -85,B 0,C 180,E1 12266.543,E2 12266.543} C_VEL
LIN {X 0,Y 333.49,Z 815.525,A -85,B 0,C 180,E1 12263.127,E2 12263.127} C_VEL
LIN {X 0,Y 328.018,Z 807.026,A -85,B 0,C 180,E1 12260.055,E2 12260.055} C_VEL
LIN {X 0,Y 324.513,Z 801.873,A -85,B 0,C 180,E1 12257.76,E2 12257.76} C_VEL
LIN {X 0,Y 321.785,Z 797.79,A -85,B 0,C 180,E1 12255.684,E2 12255.684} C_VEL
LIN {X 0,Y 318.716,Z 793.194,A -85,B 0,C 180,E1 12252.87,E2 12252.87} C_VEL
LIN {X 0,Y 315.903,Z 789.271,A -85,B 0,C 180,E1 12249.473,E2 12249.473} C_VEL
LIN {X 0,Y 315.37,Z 788.062,A -85,B 0,C 180,E1 12248.57,E2 12248.57} C_VEL
LIN {X 0,Y 313.051,Z 785.91,A -85,B 0,C 180,E1 12241.648,E2 12241.648} C_VEL
LIN {X 0,Y 313.683,Z 786.791,A -85,B 0,C 180,E1 12237.26,E2 12237.26} C_VEL
LIN {X 0,Y 315.566,Z 788.399,A -85,B 0,C 180,E1 12233.542,E2 12233.542} C_VEL
LIN {X 0,Y 317.682,Z 792.593,A -85,B 0,C 180,E1 12230.581,E2 12230.581} C_VEL
LIN {X 0,Y 320.282,Z 797.796,A -85,B 0,C 180,E1 12227.836,E2 12227.836} C_VEL
LIN {X 0,Y 323.322,Z 803.627,A -85,B 0,C 180,E1 12225.265,E2 12225.265} C_VEL
LIN {X 0,Y 327.502,Z 812.007,A -85,B 0,C 180,E1 12222.316,E2 12222.316} C_VEL
LIN {X 0,Y 332.203,Z 821.592,A -85,B 0,C 180,E1 12219.52,E2 12219.52} C_VEL
LIN {X 0,Y 337.98,Z 833.979,A -85,B 0,C 180,E1 12216.554,E2 12216.554} C_VEL
LIN {X 0,Y 340.753,Z 840.666,A -85,B 0,C 180,E1 12215.24,E2 12215.24} C_VEL
LIN {X 0,Y 327.028,Z 1017.811,A -85,B 0,C 180,E1 12211.606,E2 12211.606} C_VEL
LIN {X 0,Y 323.811,Z 1040.089,A -85,B 0,C 180,E1 12210.976,E2 12210.976} C_VEL
LIN {X 0,Y 318.856,Z 1063.588,A -85,B 0,C 180,E1 12210.113,E2 12210.113} C_VEL
LIN {X 0,Y 313.248,Z 1084.037,A -85,B 0,C 180,E1 12209.159,E2 12209.159} C_VEL
LIN {X 0,Y 306.711,Z 1103.782,A -85,B 0,C 180,E1 12207.947,E2 12207.947} C_VEL
LIN {X 0,Y 299.077,Z 1124.051,A -85,B 0,C 180,E1 12206.348,E2 12206.348} C_VEL
LIN {X 0,Y 291.174,Z 1142.929,A -85,B 0,C 180,E1 12204.47,E2 12204.47} C_VEL
LIN {X 0,Y 282.885,Z 1160.836,A -85,B 0,C 180,E1 12202.222,E2 12202.222} C_VEL
LIN {X 0,Y 273.915,Z 1178.953,A -85,B 0,C 180,E1 12199.396,E2 12199.396} C_VEL
LIN {X 0,Y 265.632,Z 1195.07,A -85,B 0,C 180,E1 12196.276,E2 12196.276} C_VEL
LIN {X 0,Y 257.798,Z 1209.847,A -85,B 0,C 180,E1 12192.743,E2 12192.743} C_VEL
LIN {X 0,Y 250.711,Z 1223.397,A -85,B 0,C 180,E1 12188.764,E2 12188.764} C_VEL
LIN {X 0,Y 244.602,Z 1235.756,A -85,B 0,C 180,E1 12184.339,E2 12184.339} C_VEL
LIN {X 0,Y 239.509,Z 1247.22,A -85,B 0,C 180,E1 12179.236,E2 12179.236} C_VEL
LIN {X 0,Y 236.114,Z 1256.621,A -85,B 0,C 180,E1 12173.986,E2 12173.986} C_VEL
LIN {X 0,Y 234.218,Z 1264.492,A -85,B 0,C 180,E1 12168.415,E2 12168.415} C_VEL
LIN {X 0,Y 233.738,Z 1269.95,A -85,B 0,C 180,E1 12163.355,E2 12163.355} C_VEL
LIN {X 0,Y 234.052,Z 1273.696,A -85,B 0,C 180,E1 12158.351,E2 12158.351} C_VEL
LIN {X 0,Y 234.533,Z 1275.534,A -85,B 0,C 180,E1 12154.401,E2 12154.401} C_VEL
LIN {X 0,Y 234.782,Z 1276.302,A -85,B 0,C 180,E1 12150.244,E2 12150.244} C_VEL
LIN {X 0,Y 234.573,Z 1275.697,A -85,B 0,C 180,E1 12146.09,E2 12146.09} C_VEL
LIN {X 0,Y 234.108,Z 1273.973,A -85,B 0,C 180,E1 12142.145,E2 12142.145} C_VEL
LIN {X 0,Y 233.754,Z 1270.808,A -85,B 0,C 180,E1 12137.651,E2 12137.651} C_VEL
LIN {X 0,Y 234.086,Z 1265.383,A -85,B 0,C 180,E1 12132.347,E2 12132.347} C_VEL
LIN {X 0,Y 235.65,Z 1258.224,A -85,B 0,C 180,E1 12127.024,E2 12127.024} C_VEL
LIN {X 0,Y 238.735,Z 1249.119,A -85,B 0,C 180,E1 12121.755,E2 12121.755} C_VEL
LIN {X 0,Y 243.23,Z 1238.581,A -85,B 0,C 180,E1 12116.858,E2 12116.858} C_VEL
LIN {X 0,Y 249.302,Z 1226.119,A -85,B 0,C 180,E1 12112.149,E2 12112.149} C_VEL
LIN {X 0,Y 256.524,Z 1212.229,A -85,B 0,C 180,E1 12107.903,E2 12107.903} C_VEL
LIN {X 0,Y 264.167,Z 1197.694,A -85,B 0,C 180,E1 12104.329,E2 12104.329} C_VEL
LIN {X 0,Y 273.094,Z 1180.448,A -85,B 0,C 180,E1 12100.886,E2 12100.886} C_VEL
LIN {X 0,Y 281.563,Z 1163.498,A -85,B 0,C 180,E1 12098.162,E2 12098.162} C_VEL
LIN {X 0,Y 289.878,Z 1145.544,A -85,B 0,C 180,E1 12095.851,E2 12095.851} C_VEL
LIN {X 0,Y 298.053,Z 1126.361,A -85,B 0,C 180,E1 12093.876,E2 12093.876} C_VEL
LIN {X 0,Y 305.641,Z 1106.609,A -85,B 0,C 180,E1 12092.262,E2 12092.262} C_VEL
LIN {X 0,Y 312.125,Z 1087.191,A -85,B 0,C 180,E1 12091.032,E2 12091.032} C_VEL
LIN {X 0,Y 318.282,Z 1065.447,A -85,B 0,C 180,E1 12089.978,E2 12089.978} C_VEL
LIN {X 0,Y 323.132,Z 1043.385,A -85,B 0,C 180,E1 12089.141,E2 12089.141} C_VEL
LIN {X 0,Y 326.545,Z 1020.938,A -85,B 0,C 180,E1 12088.485,E2 12088.485} C_VEL
LIN {X 0,Y 329.714,Z 983.192,A -85,B 0,C 180,E1 12087.671,E2 12087.671} C_VEL
LIN {X 0,Y 340.574,Z 840.116,A -85,B 0,C 180,E1 12084.73,E2 12084.73} C_VEL
LIN {X 0,Y 334.828,Z 827.341,A -85,B 0,C 180,E1 12081.963,E2 12081.963} C_VEL
LIN {X 0,Y 329.176,Z 815.496,A -85,B 0,C 180,E1 12078.828,E2 12078.828} C_VEL
LIN {X 0,Y 324.88,Z 807.006,A -85,B 0,C 180,E1 12076.034,E2 12076.034} C_VEL
LIN {X 0,Y 320.98,Z 799.242,A -85,B 0,C 180,E1 12072.96,E2 12072.96} C_VEL
LIN {X 0,Y 318.336,Z 794.211,A -85,B 0,C 180,E1 12070.404,E2 12070.404} C_VEL
LIN {X 0,Y 316.769,Z 791.004,A -85,B 0,C 180,E1 12068.531,E2 12068.531} C_VEL
LIN {X 0,Y 315.19,Z 787.954,A -85,B 0,C 180,E1 12066.191,E2 12066.191} C_VEL
LIN {X 0,Y 312.826,Z 785.622,A -85,B 0,C 180,E1 12059.267,E2 12059.267} C_VEL
LIN {X 0,Y 313.301,Z 786.392,A -85,B 0,C 180,E1 12055.24,E2 12055.24} C_VEL
LIN {X 0,Y 315.442,Z 788.314,A -85,B 0,C 180,E1 12050.881,E2 12050.881} C_VEL
LIN {X 0,Y 317.905,Z 792.459,A -85,B 0,C 180,E1 12047.65,E2 12047.65} C_VEL
LIN {X 0,Y 319.149,Z 793.931,A -85,B 0,C 180,E1 12046.41,E2 12046.41} C_VEL
LIN {X 0,Y 322.827,Z 799.405,A -85,B 0,C 180,E1 12043.259,E2 12043.259} C_VEL
LIN {X 0,Y 326.311,Z 804.64,A -85,B 0,C 180,E1 12040.814,E2 12040.814} C_VEL
LIN {X 0,Y 331.111,Z 811.819,A -85,B 0,C 180,E1 12037.968,E2 12037.968} C_VEL
LIN {X 0,Y 337.549,Z 822.461,A -85,B 0,C 180,E1 12034.704,E2 12034.704} C_VEL
LIN {X 0,Y 340.577,Z 827.762,A -85,B 0,C 180,E1 12033.33,E2 12033.33} C_VEL
LIN {X 0,Y 330.948,Z 952.581,A -85,B 0,C 180,E1 12030.757,E2 12030.757} C_VEL
LIN {X 0,Y 328.801,Z 974.371,A -85,B 0,C 180,E1 12030.085,E2 12030.085} C_VEL
LIN {X 0,Y 325.462,Z 995.527,A -85,B 0,C 180,E1 12029.184,E2 12029.184} C_VEL
LIN {X 0,Y 320.788,Z 1017.385,A -85,B 0,C 180,E1 12027.97,E2 12027.97} C_VEL
LIN {X 0,Y 315.534,Z 1036.868,A -85,B 0,C 180,E1 12026.61,E2 12026.61} C_VEL
LIN {X 0,Y 309.115,Z 1056.262,A -85,B 0,C 180,E1 12024.917,E2 12024.917} C_VEL
LIN {X 0,Y 301.977,Z 1074.735,A -85,B 0,C 180,E1 12022.933,E2 12022.933} C_VEL
LIN {X 0,Y 294.539,Z 1091.716,A -85,B 0,C 180,E1 12020.71,E2 12020.71} C_VEL
LIN {X 0,Y 286.88,Z 1107.228,A -85,B 0,C 180,E1 12018.23,E2 12018.23} C_VEL
LIN {X 0,Y 278.668,Z 1122.368,A -85,B 0,C 180,E1 12015.267,E2 12015.267} C_VEL
LIN {X 0,Y 270.644,Z 1136.113,A -85,B 0,C 180,E1 12011.964,E2 12011.964} C_VEL
LIN {X 0,Y 262.975,Z 1148.419,A -85,B 0,C 180,E1 12008.296,E2 12008.296} C_VEL
LIN {X 0,Y 255.87,Z 1159.279,A -85,B 0,C 180,E1 12004.242,E2 12004.242} C_VEL
LIN {X 0,Y 249.269,Z 1169.211,A -85,B 0,C 180,E1 11999.561,E2 11999.561} C_VEL
LIN {X 0,Y 244.244,Z 1176.904,A -85,B 0,C 180,E1 11994.938,E2 11994.938} C_VEL
LIN {X 0,Y 240.107,Z 1183.397,A -85,B 0,C 180,E1 11989.712,E2 11989.712} C_VEL
LIN {X 0,Y 237.309,Z 1188.168,A -85,B 0,C 180,E1 11984.393,E2 11984.393} C_VEL
LIN {X 0,Y 235.76,Z 1191.285,A -85,B 0,C 180,E1 11979.274,E2 11979.274} C_VEL
LIN {X 0,Y 234.999,Z 1192.957,A -85,B 0,C 180,E1 11974.148,E2 11974.148} C_VEL
LIN {X 0,Y 234.854,Z 1193.368,A -85,B 0,C 180,E1 11969.024,E2 11969.024} C_VEL
LIN {X 0,Y 235.169,Z 1192.587,A -85,B 0,C 180,E1 11964.144,E2 11964.144} C_VEL
LIN {X 0,Y 236.162,Z 1190.441,A -85,B 0,C 180,E1 11959.017,E2 11959.017} C_VEL
LIN {X 0,Y 238.021,Z 1186.994,A -85,B 0,C 180,E1 11953.905,E2 11953.905} C_VEL
LIN {X 0,Y 241.209,Z 1181.652,A -85,B 0,C 180,E1 11948.607,E2 11948.607} C_VEL
LIN {X 0,Y 245.621,Z 1174.785,A -85,B 0,C 180,E1 11943.581,E2 11943.581} C_VEL
LIN {X 0,Y 251.261,Z 1166.324,A -85,B 0,C 180,E1 11938.822,E2 11938.822} C_VEL
LIN {X 0,Y 257.902,Z 1156.365,A -85,B 0,C 180,E1 11934.443,E2 11934.443} C_VEL
LIN {X 0,Y 265.305,Z 1144.815,A -85,B 0,C 180,E1 11930.44,E2 11930.44} C_VEL
LIN {X 0,Y 273.262,Z 1131.847,A -85,B 0,C 180,E1 11926.827,E2 11926.827} C_VEL
LIN {X 0,Y 281.31,Z 1117.913,A -85,B 0,C 180,E1 11923.674,E2 11923.674} C_VEL
LIN {X 0,Y 289.425,Z 1102.429,A -85,B 0,C 180,E1 11920.84,E2 11920.84} C_VEL
LIN {X 0,Y 297.212,Z 1086.019,A -85,B 0,C 180,E1 11918.389,E2 11918.389} C_VEL
LIN {X 0,Y 304.493,Z 1068.896,A -85,B 0,C 180,E1 11916.281,E2 11916.281} C_VEL
LIN {X 0,Y 311.314,Z 1050.318,A -85,B 0,C 180,E1 11914.421,E2 11914.421} C_VEL
LIN {X 0,Y 317.269,Z 1031.143,A -85,B 0,C 180,E1 11912.861,E2 11912.861} C_VEL
LIN {X 0,Y 322.373,Z 1011.328,A -85,B 0,C 180,E1 11911.556,E2 11911.556} C_VEL
LIN {X 0,Y 326.52,Z 990.431,A -85,B 0,C 180,E1 11910.472,E2 11910.472} C_VEL
LIN {X 0,Y 329.525,Z 969.143,A -85,B 0,C 180,E1 11909.636,E2 11909.636} C_VEL
LIN {X 0,Y 331.653,Z 944.591,A -85,B 0,C 180,E1 11908.948,E2 11908.948} C_VEL
LIN {X 0,Y 337.096,Z 873.497,A -85,B 0,C 180,E1 11907.485,E2 11907.485} C_VEL
LIN {X 0,Y 337.268,Z 865.939,A -85,B 0,C 180,E1 11907.186,E2 11907.186} C_VEL
LIN {X 0,Y 336.163,Z 846.276,A -85,B 0,C 180,E1 11905.826,E2 11905.826} C_VEL
LIN {X 0,Y 336.372,Z 839.779,A -85,B 0,C 180,E1 11905.577,E2 11905.577} C_VEL
LIN {X 0,Y 336.908,Z 832.212,A -85,B 0,C 180,E1 11905.394,E2 11905.394} C_VEL
LIN {X 0,Y 330.848,Z 821.854,A -85,B 0,C 180,E1 11902.336,E2 11902.336} C_VEL
LIN {X 0,Y 325.938,Z 814.024,A -85,B 0,C 180,E1 11899.441,E2 11899.441} C_VEL
LIN {X 0,Y 322.806,Z 809.256,A -85,B 0,C 180,E1 11897.299,E2 11897.299} C_VEL
LIN {X 0,Y 320.262,Z 805.347,A -85,B 0,C 180,E1 11895.287,E2 11895.287} C_VEL
LIN {X 0,Y 317.392,Z 800.919,A -85,B 0,C 180,E1 11892.555,E2 11892.555} C_VEL
LIN {X 0,Y 314.636,Z 796.832,A -85,B 0,C 180,E1 11889.051,E2 11889.051} C_VEL
LIN {X 0,Y 314.106,Z 795.859,A -85,B 0,C 180,E1 11888.133,E2 11888.133} C_VEL
LIN {X 0,Y 312.077,Z 793.852,A -85,B 0,C 180,E1 11881.653,E2 11881.653} C_VEL
LIN {X 0,Y 312.707,Z 794.749,A -85,B 0,C 180,E1 11877.251,E2 11877.251} C_VEL
LIN {X 0,Y 314.414,Z 796.222,A -85,B 0,C 180,E1 11873.793,E2 11873.793} C_VEL
LIN {X 0,Y 316.385,Z 800.301,A -85,B 0,C 180,E1 11870.909,E2 11870.909} C_VEL
LIN {X 0,Y 318.896,Z 805.52,A -85,B 0,C 180,E1 11868.149,E2 11868.149} C_VEL
LIN {X 0,Y 321.736,Z 811.254,A -85,B 0,C 180,E1 11865.651,E2 11865.651} C_VEL
LIN {X 0,Y 325.484,Z 819.013,A -85,B 0,C 180,E1 11862.895,E2 11862.895} C_VEL
LIN {X 0,Y 330.099,Z 828.752,A -85,B 0,C 180,E1 11860.031,E2 11860.031} C_VEL
LIN {X 0,Y 335.543,Z 840.933,A -85,B 0,C 180,E1 11857.116,E2 11857.116} C_VEL
LIN {X 0,Y 336.996,Z 844.643,A -85,B 0,C 180,E1 11856.385,E2 11856.385} C_VEL
LIN {X 0,Y 323.249,Z 1016.4,A -85,B 0,C 180,E1 11852.87,E2 11852.87} C_VEL
LIN {X 0,Y 319.942,Z 1038.746,A -85,B 0,C 180,E1 11852.243,E2 11852.243} C_VEL
LIN {X 0,Y 314.894,Z 1062.164,A -85,B 0,C 180,E1 11851.393,E2 11851.393} C_VEL
LIN {X 0,Y 309.159,Z 1082.609,A -85,B 0,C 180,E1 11850.453,E2 11850.453} C_VEL
LIN {X 0,Y 302.453,Z 1102.345,A -85,B 0,C 180,E1 11849.259,E2 11849.259} C_VEL
LIN {X 0,Y 294.599,Z 1122.605,A -85,B 0,C 180,E1 11847.679,E2 11847.679} C_VEL
LIN {X 0,Y 286.384,Z 1141.613,A -85,B 0,C 180,E1 11845.799,E2 11845.799} C_VEL
LIN {X 0,Y 277.893,Z 1159.327,A -85,B 0,C 180,E1 11843.583,E2 11843.583} C_VEL
LIN {X 0,Y 268.544,Z 1177.479,A -85,B 0,C 180,E1 11840.752,E2 11840.752} C_VEL
LIN {X 0,Y 259.888,Z 1193.588,A -85,B 0,C 180,E1 11837.617,E2 11837.617} C_VEL
LIN {X 0,Y 251.585,Z 1208.53,A -85,B 0,C 180,E1 11834.001,E2 11834.001} C_VEL
LIN {X 0,Y 243.797,Z 1222.602,A -85,B 0,C 180,E1 11829.774,E2 11829.774} C_VEL
LIN {X 0,Y 237.074,Z 1235.416,A -85,B 0,C 180,E1 11824.999,E2 11824.999} C_VEL
LIN {X 0,Y 231.938,Z 1246.352,A -85,B 0,C 180,E1 11819.948,E2 11819.948} C_VEL
LIN {X 0,Y 228.36,Z 1255.554,A -85,B 0,C 180,E1 11814.578,E2 11814.578} C_VEL
LIN {X 0,Y 226.327,Z 1263.337,A -85,B 0,C 180,E1 11808.813,E2 11808.813} C_VEL
LIN {X 0,Y 225.794,Z 1268.758,A -85,B 0,C 180,E1 11803.573,E2 11803.573} C_VEL
LIN {X 0,Y 226.109,Z 1272.279,A -85,B 0,C 180,E1 11798.647,E2 11798.647} C_VEL
LIN {X 0,Y 226.637,Z 1274.183,A -85,B 0,C 180,E1 11794.411,E2 11794.411} C_VEL
LIN {X 0,Y 226.902,Z 1274.912,A -85,B 0,C 180,E1 11790.252,E2 11790.252} C_VEL
LIN {X 0,Y 226.693,Z 1274.383,A -85,B 0,C 180,E1 11786.207,E2 11786.207} C_VEL
LIN {X 0,Y 226.166,Z 1272.557,A -85,B 0,C 180,E1 11781.867,E2 11781.867} C_VEL
LIN {X 0,Y 225.808,Z 1269.371,A -85,B 0,C 180,E1 11777.209,E2 11777.209} C_VEL
LIN {X 0,Y 226.225,Z 1263.924,A -85,B 0,C 180,E1 11771.712,E2 11771.712} C_VEL
LIN {X 0,Y 227.986,Z 1256.749,A -85,B 0,C 180,E1 11766.205,E2 11766.205} C_VEL
LIN {X 0,Y 231.359,Z 1247.634,A -85,B 0,C 180,E1 11760.769,E2 11760.769} C_VEL
LIN {X 0,Y 236.206,Z 1237.09,A -85,B 0,C 180,E1 11755.738,E2 11755.738} C_VEL
LIN {X 0,Y 242.687,Z 1224.627,A -85,B 0,C 180,E1 11750.925,E2 11750.925} C_VEL
LIN {X 0,Y 250.329,Z 1210.738,A -85,B 0,C 180,E1 11746.609,E2 11746.609} C_VEL
LIN {X 0,Y 258.678,Z 1195.635,A -85,B 0,C 180,E1 11742.865,E2 11742.865} C_VEL
LIN {X 0,Y 267.686,Z 1178.967,A -85,B 0,C 180,E1 11739.53,E2 11739.53} C_VEL
LIN {X 0,Y 276.545,Z 1161.926,A -85,B 0,C 180,E1 11736.792,E2 11736.792} C_VEL
LIN {X 0,Y 285.114,Z 1144.081,A -85,B 0,C 180,E1 11734.504,E2 11734.504} C_VEL
LIN {X 0,Y 293.513,Z 1124.988,A -85,B 0,C 180,E1 11732.551,E2 11732.551} C_VEL
LIN {X 0,Y 300.995,Z 1106.184,A -85,B 0,C 180,E1 11731.018,E2 11731.018} C_VEL
LIN {X 0,Y 308.013,Z 1085.748,A -85,B 0,C 180,E1 11729.736,E2 11729.736} C_VEL
LIN {X 0,Y 314.318,Z 1063.97,A -85,B 0,C 180,E1 11728.696,E2 11728.696} C_VEL
LIN {X 0,Y 319.237,Z 1042.073,A -85,B 0,C 180,E1 11727.873,E2 11727.873} C_VEL
LIN {X 0,Y 322.731,Z 1019.655,A -85,B 0,C 180,E1 11727.224,E2 11727.224} C_VEL
LIN {X 0,Y 325.928,Z 982.97,A -85,B 0,C 180,E1 11726.432,E2 11726.432} C_VEL
LIN {X 0,Y 336.846,Z 844.157,A -85,B 0,C 180,E1 11723.6,E2 11723.6} C_VEL
LIN {X 0,Y 331.202,Z 831.331,A -85,B 0,C 180,E1 11720.683,E2 11720.683} C_VEL
LIN {X 0,Y 326.415,Z 821.196,A -85,B 0,C 180,E1 11717.837,E2 11717.837} C_VEL
LIN {X 0,Y 322.895,Z 813.918,A -85,B 0,C 180,E1 11715.398,E2 11715.398} C_VEL
LIN {X 0,Y 319.276,Z 806.434,A -85,B 0,C 180,E1 11712.387,E2 11712.387} C_VEL
LIN {X 0,Y 316.772,Z 801.435,A -85,B 0,C 180,E1 11709.813,E2 11709.813} C_VEL
LIN {X 0,Y 315.432,Z 798.582,A -85,B 0,C 180,E1 11708.109,E2 11708.109} C_VEL
LIN {X 0,Y 314.098,Z 795.846,A -85,B 0,C 180,E1 11706.03,E2 11706.03} C_VEL
LIN {X 0,Y 311.851,Z 793.564,A -85,B 0,C 180,E1 11699.265,E2 11699.265} C_VEL
LIN {X 0,Y 312.327,Z 794.352,A -85,B 0,C 180,E1 11695.225,E2 11695.225} C_VEL
LIN {X 0,Y 314.289,Z 796.154,A -85,B 0,C 180,E1 11691.124,E2 11691.124} C_VEL
LIN {X 0,Y 316.767,Z 800.352,A -85,B 0,C 180,E1 11687.79,E2 11687.79} C_VEL
LIN {X 0,Y 317.89,Z 801.824,A -85,B 0,C 180,E1 11686.633,E2 11686.633} C_VEL
LIN {X 0,Y 321.386,Z 807.156,A -85,B 0,C 180,E1 11683.554,E2 11683.554} C_VEL
LIN {X 0,Y 324.67,Z 812.219,A -85,B 0,C 180,E1 11681.18,E2 11681.18} C_VEL
LIN {X 0,Y 329.22,Z 819.25,A -85,B 0,C 180,E1 11678.392,E2 11678.392} C_VEL
LIN {X 0,Y 335.935,Z 830.592,A -85,B 0,C 180,E1 11674.904,E2 11674.904} C_VEL
LIN {X 0,Y 336.828,Z 832.471,A -85,B 0,C 180,E1 11674.467,E2 11674.467} C_VEL
LIN {X 0,Y 327.215,Z 953.367,A -85,B 0,C 180,E1 11671.981,E2 11671.981} C_VEL
LIN {X 0,Y 325.013,Z 975.137,A -85,B 0,C 180,E1 11671.313,E2 11671.313} C_VEL
LIN {X 0,Y 321.595,Z 996.4,A -85,B 0,C 180,E1 11670.416,E2 11670.416} C_VEL
LIN {X 0,Y 317.112,Z 1017.112,A -85,B 0,C 180,E1 11669.283,E2 11669.283} C_VEL
LIN {X 0,Y 311.582,Z 1037.209,A -85,B 0,C 180,E1 11667.902,E2 11667.902} C_VEL
LIN {X 0,Y 305.271,Z 1055.927,A -85,B 0,C 180,E1 11666.295,E2 11666.295} C_VEL
LIN {X 0,Y 297.537,Z 1075.551,A -85,B 0,C 180,E1 11664.217,E2 11664.217} C_VEL
LIN {X 0,Y 289.894,Z 1092.535,A -85,B 0,C 180,E1 11662.007,E2 11662.007} C_VEL
LIN {X 0,Y 281.672,Z 1108.628,A -85,B 0,C 180,E1 11659.431,E2 11659.431} C_VEL
LIN {X 0,Y 273.149,Z 1123.769,A -85,B 0,C 180,E1 11656.448,E2 11656.448} C_VEL
LIN {X 0,Y 264.793,Z 1137.517,A -85,B 0,C 180,E1 11653.113,E2 11653.113} C_VEL
LIN {X 0,Y 256.782,Z 1149.824,A -85,B 0,C 180,E1 11649.395,E2 11649.395} C_VEL
LIN {X 0,Y 249.327,Z 1160.686,A -85,B 0,C 180,E1 11645.272,E2 11645.272} C_VEL
LIN {X 0,Y 242.37,Z 1170.618,A -85,B 0,C 180,E1 11640.491,E2 11640.491} C_VEL
LIN {X 0,Y 237.048,Z 1178.31,A -85,B 0,C 180,E1 11635.749,E2 11635.749} C_VEL
LIN {X 0,Y 232.632,Z 1184.802,A -85,B 0,C 180,E1 11630.373,E2 11630.373} C_VEL
LIN {X 0,Y 229.604,Z 1189.618,A -85,B 0,C 180,E1 11624.816,E2 11624.816} C_VEL
LIN {X 0,Y 227.898,Z 1192.776,A -85,B 0,C 180,E1 11619.342,E2 11619.342} C_VEL
LIN {X 0,Y 227.134,Z 1194.348,A -85,B 0,C 180,E1 11614.292,E2 11614.292} C_VEL
LIN {X 0,Y 226.977,Z 1194.758,A -85,B 0,C 180,E1 11608.99,E2 11608.99} C_VEL
LIN {X 0,Y 227.318,Z 1193.98,A -85,B 0,C 180,E1 11603.941,E2 11603.941} C_VEL
LIN {X 0,Y 228.394,Z 1191.837,A -85,B 0,C 180,E1 11598.639,E2 11598.639} C_VEL
LIN {X 0,Y 230.399,Z 1188.395,A -85,B 0,C 180,E1 11593.357,E2 11593.357} C_VEL
LIN {X 0,Y 233.627,Z 1183.324,A -85,B 0,C 180,E1 11588.141,E2 11588.141} C_VEL
LIN {X 0,Y 238.436,Z 1176.3,A -85,B 0,C 180,E1 11582.802,E2 11582.802} C_VEL
LIN {X 0,Y 244.135,Z 1168.244,A -85,B 0,C 180,E1 11578.109,E2 11578.109} C_VEL
LIN {X 0,Y 251.084,Z 1158.295,A -85,B 0,C 180,E1 11573.607,E2 11573.607} C_VEL
LIN {X 0,Y 258.789,Z 1146.866,A -85,B 0,C 180,E1 11569.529,E2 11569.529} C_VEL
LIN {X 0,Y 267.046,Z 1134.037,A -85,B 0,C 180,E1 11565.862,E2 11565.862} C_VEL
LIN {X 0,Y 275.637,Z 1119.78,A -85,B 0,C 180,E1 11562.579,E2 11562.579} C_VEL
LIN {X 0,Y 284.032,Z 1104.348,A -85,B 0,C 180,E1 11559.723,E2 11559.723} C_VEL
LIN {X 0,Y 292.373,Z 1087.408,A -85,B 0,C 180,E1 11557.175,E2 11557.175} C_VEL
LIN {X 0,Y 299.892,Z 1070.283,A -85,B 0,C 180,E1 11555.066,E2 11555.066} C_VEL
LIN {X 0,Y 306.705,Z 1052.308,A -85,B 0,C 180,E1 11553.263,E2 11553.263} C_VEL
LIN {X 0,Y 313.032,Z 1032.635,A -85,B 0,C 180,E1 11551.657,E2 11551.657} C_VEL
LIN {X 0,Y 318.296,Z 1012.818,A -85,B 0,C 180,E1 11550.354,E2 11550.354} C_VEL
LIN {X 0,Y 322.593,Z 991.811,A -85,B 0,C 180,E1 11549.265,E2 11549.265} C_VEL
LIN {X 0,Y 325.697,Z 970.49,A -85,B 0,C 180,E1 11548.427,E2 11548.427} C_VEL
LIN {X 0,Y 327.905,Z 945.836,A -85,B 0,C 180,E1 11547.735,E2 11547.735} C_VEL
LIN {X 0,Y 336.372,Z 839.779,A -85,B 0,C 180,E1 11545.577,E2 11545.577} C_VEL
LIN {X 0,Y 336.185,Z 837.028,A -85,B 0,C 180,E1 11545.366,E2 11545.366} C_VEL
LIN {X 0,Y 335.231,Z 834.6,A -85,B 0,C 180,E1 11544.873,E2 11544.873} C_VEL
LIN {X 0,Y 333.165,Z 832.604,A -85,B 0,C 180,E1 11543.939,E2 11543.939} C_VEL
LIN {X 0,Y 329.672,Z 830.273,A -85,B 0,C 180,E1 11542.305,E2 11542.305} C_VEL
LIN {X 0,Y 329.181,Z 829.619,A -85,B 0,C 180,E1 11542.043,E2 11542.043} C_VEL
LIN {X 0,Y 324.156,Z 821.394,A -85,B 0,C 180,E1 11538.991,E2 11538.991} C_VEL
LIN {X 0,Y 321.006,Z 816.469,A -85,B 0,C 180,E1 11536.745,E2 11536.745} C_VEL
LIN {X 0,Y 318.673,Z 812.799,A -85,B 0,C 180,E1 11534.816,E2 11534.816} C_VEL
LIN {X 0,Y 316.078,Z 808.642,A -85,B 0,C 180,E1 11532.237,E2 11532.237} C_VEL
LIN {X 0,Y 313.436,Z 804.526,A -85,B 0,C 180,E1 11528.716,E2 11528.716} C_VEL
LIN {X 0,Y 312.979,Z 803.724,A -85,B 0,C 180,E1 11527.896,E2 11527.896} C_VEL
LIN {X 0,Y 311.098,Z 801.779,A -85,B 0,C 180,E1 11521.474,E2 11521.474} C_VEL
LIN {X 0,Y 311.859,Z 802.849,A -85,B 0,C 180,E1 11516.876,E2 11516.876} C_VEL
LIN {X 0,Y 313.315,Z 804.177,A -85,B 0,C 180,E1 11513.955,E2 11513.955} C_VEL
LIN {X 0,Y 315.098,Z 808.007,A -85,B 0,C 180,E1 11511.239,E2 11511.239} C_VEL
LIN {X 0,Y 317.521,Z 813.24,A -85,B 0,C 180,E1 11508.466,E2 11508.466} C_VEL
LIN {X 0,Y 320.372,Z 819.351,A -85,B 0,C 180,E1 11505.865,E2 11505.865} C_VEL
LIN {X 0,Y 323.56,Z 826.158,A -85,B 0,C 180,E1 11503.437,E2 11503.437} C_VEL
LIN {X 0,Y 327.949,Z 835.768,A -85,B 0,C 180,E1 11500.591,E2 11500.591} C_VEL
LIN {X 0,Y 333.141,Z 847.878,A -85,B 0,C 180,E1 11497.687,E2 11497.687} C_VEL
LIN {X 0,Y 333.353,Z 848.9,A -85,B 0,C 180,E1 11497.55,E2 11497.55} C_VEL
LIN {X 0,Y 319.631,Z 1014.989,A -85,B 0,C 180,E1 11494.165,E2 11494.165} C_VEL
LIN {X 0,Y 316.254,Z 1037.284,A -85,B 0,C 180,E1 11493.545,E2 11493.545} C_VEL
LIN {X 0,Y 311.091,Z 1060.741,A -85,B 0,C 180,E1 11492.704,E2 11492.704} C_VEL
LIN {X 0,Y 305.233,Z 1081.181,A -85,B 0,C 180,E1 11491.78,E2 11491.78} C_VEL
LIN {X 0,Y 298.357,Z 1100.908,A -85,B 0,C 180,E1 11490.609,E2 11490.609} C_VEL
LIN {X 0,Y 290.286,Z 1121.158,A -85,B 0,C 180,E1 11489.051,E2 11489.051} C_VEL
LIN {X 0,Y 281.886,Z 1140.019,A -85,B 0,C 180,E1 11487.206,E2 11487.206} C_VEL
LIN {X 0,Y 272.936,Z 1158.072,A -85,B 0,C 180,E1 11484.958,E2 11484.958} C_VEL
LIN {X 0,Y 263.337,Z 1176.007,A -85,B 0,C 180,E1 11482.16,E2 11482.16} C_VEL
LIN {X 0,Y 254.298,Z 1192.107,A -85,B 0,C 180,E1 11479.016,E2 11479.016} C_VEL
LIN {X 0,Y 245.686,Z 1206.877,A -85,B 0,C 180,E1 11475.411,E2 11475.411} C_VEL
LIN {X 0,Y 237.767,Z 1220.418,A -85,B 0,C 180,E1 11471.315,E2 11471.315} C_VEL
LIN {X 0,Y 230.847,Z 1232.777,A -85,B 0,C 180,E1 11466.705,E2 11466.705} C_VEL
LIN {X 0,Y 225.076,Z 1243.979,A -85,B 0,C 180,E1 11461.47,E2 11461.47} C_VEL
LIN {X 0,Y 221.068,Z 1253.258,A -85,B 0,C 180,E1 11456.021,E2 11456.021} C_VEL
LIN {X 0,Y 218.704,Z 1260.959,A -85,B 0,C 180,E1 11450.331,E2 11450.331} C_VEL
LIN {X 0,Y 217.891,Z 1266.565,A -85,B 0,C 180,E1 11444.89,E2 11444.89} C_VEL
LIN {X 0,Y 218.102,Z 1270.565,A -85,B 0,C 180,E1 11439.499,E2 11439.499} C_VEL
LIN {X 0,Y 218.664,Z 1272.642,A -85,B 0,C 180,E1 11434.984,E2 11434.984} C_VEL
LIN {X 0,Y 219.009,Z 1273.445,A -85,B 0,C 180,E1 11431.046,E2 11431.046} C_VEL
LIN {X 0,Y 218.89,Z 1273.221,A -85,B 0,C 180,E1 11427.12,E2 11427.12} C_VEL
LIN {X 0,Y 218.344,Z 1271.715,A -85,B 0,C 180,E1 11422.633,E2 11422.633} C_VEL
LIN {X 0,Y 217.9,Z 1268.715,A -85,B 0,C 180,E1 11417.786,E2 11417.786} C_VEL
LIN {X 0,Y 218.186,Z 1263.677,A -85,B 0,C 180,E1 11412.12,E2 11412.12} C_VEL
LIN {X 0,Y 219.746,Z 1257.127,A -85,B 0,C 180,E1 11406.681,E2 11406.681} C_VEL
LIN {X 0,Y 223.101,Z 1248.247,A -85,B 0,C 180,E1 11400.916,E2 11400.916} C_VEL
LIN {X 0,Y 228.093,Z 1237.895,A -85,B 0,C 180,E1 11395.566,E2 11395.566} C_VEL
LIN {X 0,Y 234.67,Z 1225.822,A -85,B 0,C 180,E1 11390.593,E2 11390.593} C_VEL
LIN {X 0,Y 242.441,Z 1212.288,A -85,B 0,C 180,E1 11386.145,E2 11386.145} C_VEL
LIN {X 0,Y 251.654,Z 1196.529,A -85,B 0,C 180,E1 11382.016,E2 11382.016} C_VEL
LIN {X 0,Y 260.716,Z 1180.663,A -85,B 0,C 180,E1 11378.69,E2 11378.69} C_VEL
LIN {X 0,Y 270.059,Z 1163.442,A -85,B 0,C 180,E1 11375.827,E2 11375.827} C_VEL
LIN {X 0,Y 279.159,Z 1145.391,A -85,B 0,C 180,E1 11373.435,E2 11373.435} C_VEL
LIN {X 0,Y 287.788,Z 1126.791,A -85,B 0,C 180,E1 11371.47,E2 11371.47} C_VEL
LIN {X 0,Y 295.376,Z 1108.453,A -85,B 0,C 180,E1 11369.941,E2 11369.941} C_VEL
LIN {X 0,Y 302.931,Z 1087.682,A -85,B 0,C 180,E1 11368.593,E2 11368.593} C_VEL
LIN {X 0,Y 309.521,Z 1066.318,A -85,B 0,C 180,E1 11367.539,E2 11367.539} C_VEL
LIN {X 0,Y 314.808,Z 1044.241,A -85,B 0,C 180,E1 11366.691,E2 11366.691} C_VEL
LIN {X 0,Y 318.573,Z 1021.99,A -85,B 0,C 180,E1 11366.028,E2 11366.028} C_VEL
LIN {X 0,Y 321.438,Z 993.521,A -85,B 0,C 180,E1 11365.386,E2 11365.386} C_VEL
LIN {X 0,Y 333.206,Z 848.288,A -85,B 0,C 180,E1 11362.43,E2 11362.43} C_VEL
LIN {X 0,Y 328.075,Z 836.306,A -85,B 0,C 180,E1 11359.587,E2 11359.587} C_VEL
LIN {X 0,Y 323.82,Z 826.989,A -85,B 0,C 180,E1 11356.872,E2 11356.872} C_VEL
LIN {X 0,Y 320.676,Z 820.257,A -85,B 0,C 180,E1 11354.536,E2 11354.536} C_VEL
LIN {X 0,Y 317.513,Z 813.443,A -85,B 0,C 180,E1 11351.719,E2 11351.719} C_VEL
LIN {X 0,Y 314.58,Z 806.944,A -85,B 0,C 180,E1 11348.315,E2 11348.315} C_VEL
LIN {X 0,Y 312.894,Z 803.673,A -85,B 0,C 180,E1 11345.685,E2 11345.685} C_VEL
LIN {X 0,Y 310.87,Z 801.487,A -85,B 0,C 180,E1 11339.078,E2 11339.078} C_VEL
LIN {X 0,Y 311.465,Z 802.456,A -85,B 0,C 180,E1 11334.843,E2 11334.843} C_VEL
LIN {X 0,Y 313.191,Z 804.129,A -85,B 0,C 180,E1 11331.278,E2 11331.278} C_VEL
LIN {X 0,Y 315.799,Z 808.418,A -85,B 0,C 180,E1 11327.752,E2 11327.752} C_VEL
LIN {X 0,Y 317.064,Z 810.508,A -85,B 0,C 180,E1 11326.412,E2 11326.412} C_VEL
LIN {X 0,Y 319.849,Z 814.714,A -85,B 0,C 180,E1 11323.939,E2 11323.939} C_VEL
LIN {X 0,Y 323.166,Z 819.999,A -85,B 0,C 180,E1 11321.464,E2 11321.464} C_VEL
LIN {X 0,Y 327.411,Z 826.79,A -85,B 0,C 180,E1 11318.784,E2 11318.784} C_VEL
LIN {X 0,Y 333.231,Z 836.917,A -85,B 0,C 180,E1 11315.637,E2 11315.637} C_VEL
LIN {X 0,Y 323.631,Z 954.204,A -85,B 0,C 180,E1 11313.232,E2 11313.232} C_VEL
LIN {X 0,Y 321.373,Z 975.943,A -85,B 0,C 180,E1 11312.568,E2 11312.568} C_VEL
LIN {X 0,Y 317.85,Z 997.43,A -85,B 0,C 180,E1 11311.67,E2 11311.67} C_VEL
LIN {X 0,Y 313.358,Z 1017.778,A -85,B 0,C 180,E1 11310.568,E2 11310.568} C_VEL
LIN {X 0,Y 307.79,Z 1037.514,A -85,B 0,C 180,E1 11309.227,E2 11309.227} C_VEL
LIN {X 0,Y 301.291,Z 1056.457,A -85,B 0,C 180,E1 11307.624,E2 11307.624} C_VEL
LIN {X 0,Y 293.989,Z 1074.716,A -85,B 0,C 180,E1 11305.733,E2 11305.733} C_VEL
LIN {X 0,Y 285.995,Z 1092.085,A -85,B 0,C 180,E1 11303.521,E2 11303.521} C_VEL
LIN {X 0,Y 277.541,Z 1108.274,A -85,B 0,C 180,E1 11300.98,E2 11300.98} C_VEL
LIN {X 0,Y 268.83,Z 1123.426,A -85,B 0,C 180,E1 11298.059,E2 11298.059} C_VEL
LIN {X 0,Y 260.045,Z 1137.462,A -85,B 0,C 180,E1 11294.717,E2 11294.717} C_VEL
LIN {X 0,Y 251.479,Z 1150.055,A -85,B 0,C 180,E1 11290.937,E2 11290.937} C_VEL
LIN {X 0,Y 243.253,Z 1161.566,A -85,B 0,C 180,E1 11286.583,E2 11286.583} C_VEL
LIN {X 0,Y 236.181,Z 1171.194,A -85,B 0,C 180,E1 11281.949,E2 11281.949} C_VEL
LIN {X 0,Y 230.155,Z 1179.356,A -85,B 0,C 180,E1 11276.859,E2 11276.859} C_VEL
LIN {X 0,Y 225.548,Z 1185.672,A -85,B 0,C 180,E1 11271.588,E2 11271.588} C_VEL
LIN {X 0,Y 222.089,Z 1190.792,A -85,B 0,C 180,E1 11265.671,E2 11265.671} C_VEL
LIN {X 0,Y 220.236,Z 1193.979,A -85,B 0,C 180,E1 11260.198,E2 11260.198} C_VEL
LIN {X 0,Y 219.294,Z 1195.682,A -85,B 0,C 180,E1 11254.707,E2 11254.707} C_VEL
LIN {X 0,Y 219.094,Z 1196.169,A -85,B 0,C 180,E1 11249.216,E2 11249.216} C_VEL
LIN {X 0,Y 219.436,Z 1195.428,A -85,B 0,C 180,E1 11243.985,E2 11243.985} C_VEL
LIN {X 0,Y 220.654,Z 1193.203,A -85,B 0,C 180,E1 11238.175,E2 11238.175} C_VEL
LIN {X 0,Y 222.938,Z 1189.572,A -85,B 0,C 180,E1 11232.514,E2 11232.514} C_VEL
LIN {X 0,Y 226.456,Z 1184.461,A -85,B 0,C 180,E1 11227.137,E2 11227.137} C_VEL
LIN {X 0,Y 231.532,Z 1177.496,A -85,B 0,C 180,E1 11221.76,E2 11221.76} C_VEL
LIN {X 0,Y 237.85,Z 1169.021,A -85,B 0,C 180,E1 11216.778,E2 11216.778} C_VEL
LIN {X 0,Y 245.125,Z 1159.171,A -85,B 0,C 180,E1 11212.278,E2 11212.278} C_VEL
LIN {X 0,Y 253.25,Z 1147.616,A -85,B 0,C 180,E1 11208.148,E2 11208.148} C_VEL
LIN {X 0,Y 261.911,Z 1134.643,A -85,B 0,C 180,E1 11204.45,E2 11204.45} C_VEL
LIN {X 0,Y 270.608,Z 1120.703,A -85,B 0,C 180,E1 11201.246,E2 11201.246} C_VEL
LIN {X 0,Y 279.333,Z 1105.215,A -85,B 0,C 180,E1 11198.383,E2 11198.383} C_VEL
LIN {X 0,Y 287.669,Z 1088.798,A -85,B 0,C 180,E1 11195.922,E2 11195.922} C_VEL
LIN {X 0,Y 295.43,Z 1071.67,A -85,B 0,C 180,E1 11193.814,E2 11193.814} C_VEL
LIN {X 0,Y 302.454,Z 1053.693,A -85,B 0,C 180,E1 11192.014,E2 11192.014} C_VEL
LIN {X 0,Y 308.969,Z 1034.019,A -85,B 0,C 180,E1 11190.413,E2 11190.413} C_VEL
LIN {X 0,Y 314.368,Z 1014.284,A -85,B 0,C 180,E1 11189.119,E2 11189.119} C_VEL
LIN {X 0,Y 318.761,Z 993.446,A -85,B 0,C 180,E1 11188.04,E2 11188.04} C_VEL
LIN {X 0,Y 321.988,Z 972.057,A -85,B 0,C 180,E1 11187.198,E2 11187.198} C_VEL
LIN {X 0,Y 324.26,Z 947.709,A -85,B 0,C 180,E1 11186.509,E2 11186.509} C_VEL
LIN {X 0,Y 333.369,Z 837.008,A -85,B 0,C 180,E1 11184.262,E2 11184.262} C_VEL
LIN {X 0,Y 329.181,Z 829.619,A -85,B 0,C 180,E1 11182.043,E2 11182.043} C_VEL
LIN {X 0,Y 326.891,Z 827.298,A -85,B 0,C 180,E1 11180.812,E2 11180.812} C_VEL
LIN {X 0,Y 320.108,Z 824.669,A -85,B 0,C 180,E1 11176.84,E2 11176.84} C_VEL
LIN {X 0,Y 319.114,Z 823.478,A -85,B 0,C 180,E1 11176.086,E2 11176.086} C_VEL
LIN {X 0,Y 317.097,Z 820.23,A -85,B 0,C 180,E1 11174.331,E2 11174.331} C_VEL
LIN {X 0,Y 314.774,Z 816.362,A -85,B 0,C 180,E1 11171.916,E2 11171.916} C_VEL
LIN {X 0,Y 312.194,Z 812.063,A -85,B 0,C 180,E1 11168.271,E2 11168.271} C_VEL
LIN {X 0,Y 310.19,Z 809.869,A -85,B 0,C 180,E1 11162.587,E2 11162.587} C_VEL
LIN {X 0,Y 310.295,Z 810.054,A -85,B 0,C 180,E1 11159.077,E2 11159.077} C_VEL
LIN {X 0,Y 312.174,Z 811.994,A -85,B 0,C 180,E1 11154.21,E2 11154.21} C_VEL
LIN {X 0,Y 313.821,Z 815.711,A -85,B 0,C 180,E1 11151.573,E2 11151.573} C_VEL
LIN {X 0,Y 316.156,Z 820.958,A -85,B 0,C 180,E1 11148.785,E2 11148.785} C_VEL
LIN {X 0,Y 319.437,Z 828.329,A -85,B 0,C 180,E1 11145.73,E2 11145.73} C_VEL
LIN {X 0,Y 323.117,Z 836.505,A -85,B 0,C 180,E1 11142.951,E2 11142.951} C_VEL
LIN {X 0,Y 328.122,Z 848.26,A -85,B 0,C 180,E1 11139.766,E2 11139.766} C_VEL
LIN {X 0,Y 329.884,Z 852.77,A -85,B 0,C 180,E1 11138.747,E2 11138.747} C_VEL
LIN {X 0,Y 316.181,Z 1013.578,A -85,B 0,C 180,E1 11135.488,E2 11135.488} C_VEL
LIN {X 0,Y 312.725,Z 1035.865,A -85,B 0,C 180,E1 11134.876,E2 11134.876} C_VEL
LIN {X 0,Y 307.457,Z 1059.319,A -85,B 0,C 180,E1 11134.048,E2 11134.048} C_VEL
LIN {X 0,Y 301.476,Z 1079.754,A -85,B 0,C 180,E1 11133.141,E2 11133.141} C_VEL
LIN {X 0,Y 294.434,Z 1099.473,A -85,B 0,C 180,E1 11131.994,E2 11131.994} C_VEL
LIN {X 0,Y 286.146,Z 1119.713,A -85,B 0,C 180,E1 11130.463,E2 11130.463} C_VEL
LIN {X 0,Y 277.496,Z 1138.564,A -85,B 0,C 180,E1 11128.641,E2 11128.641} C_VEL
LIN {X 0,Y 268.249,Z 1156.608,A -85,B 0,C 180,E1 11126.412,E2 11126.412} C_VEL
LIN {X 0,Y 258.3,Z 1174.537,A -85,B 0,C 180,E1 11123.622,E2 11123.622} C_VEL
LIN {X 0,Y 248.872,Z 1190.628,A -85,B 0,C 180,E1 11120.475,E2 11120.475} C_VEL
LIN {X 0,Y 239.84,Z 1205.391,A -85,B 0,C 180,E1 11116.847,E2 11116.847} C_VEL
LIN {X 0,Y 231.496,Z 1218.931,A -85,B 0,C 180,E1 11112.694,E2 11112.694} C_VEL
LIN {X 0,Y 224.126,Z 1231.287,A -85,B 0,C 180,E1 11107.997,E2 11107.997} C_VEL
LIN {X 0,Y 218.05,Z 1242.244,A -85,B 0,C 180,E1 11102.756,E2 11102.756} C_VEL
LIN {X 0,Y 213.566,Z 1251.78,A -85,B 0,C 180,E1 11097.008,E2 11097.008} C_VEL
LIN {X 0,Y 210.937,Z 1259.494,A -85,B 0,C 180,E1 11091.115,E2 11091.115} C_VEL
LIN {X 0,Y 209.973,Z 1265.118,A -85,B 0,C 180,E1 11085.465,E2 11085.465} C_VEL
LIN {X 0,Y 210.147,Z 1269.141,A -85,B 0,C 180,E1 11079.862,E2 11079.862} C_VEL
LIN {X 0,Y 210.75,Z 1271.24,A -85,B 0,C 180,E1 11075.172,E2 11075.172} C_VEL
LIN {X 0,Y 211.129,Z 1272.054,A -85,B 0,C 180,E1 11071.085,E2 11071.085} C_VEL
LIN {X 0,Y 210.994,Z 1271.825,A -85,B 0,C 180,E1 11067.012,E2 11067.012} C_VEL
LIN {X 0,Y 210.4,Z 1270.301,A -85,B 0,C 180,E1 11062.354,E2 11062.354} C_VEL
LIN {X 0,Y 209.951,Z 1267.3,A -85,B 0,C 180,E1 11057.346,E2 11057.346} C_VEL
LIN {X 0,Y 210.283,Z 1262.521,A -85,B 0,C 180,E1 11051.711,E2 11051.711} C_VEL
LIN {X 0,Y 212.104,Z 1255.653,A -85,B 0,C 180,E1 11045.789,E2 11045.789} C_VEL
LIN {X 0,Y 215.686,Z 1246.977,A -85,B 0,C 180,E1 11039.958,E2 11039.958} C_VEL
LIN {X 0,Y 220.916,Z 1236.898,A -85,B 0,C 180,E1 11034.554,E2 11034.554} C_VEL
LIN {X 0,Y 227.811,Z 1224.962,A -85,B 0,C 180,E1 11029.492,E2 11029.492} C_VEL
LIN {X 0,Y 235.961,Z 1211.558,A -85,B 0,C 180,E1 11024.958,E2 11024.958} C_VEL
LIN {X 0,Y 245.026,Z 1196.85,A -85,B 0,C 180,E1 11020.984,E2 11020.984} C_VEL
LIN {X 0,Y 254.648,Z 1180.768,A -85,B 0,C 180,E1 11017.523,E2 11017.523} C_VEL
LIN {X 0,Y 264.151,Z 1163.982,A -85,B 0,C 180,E1 11014.675,E2 11014.675} C_VEL
LIN {X 0,Y 273.996,Z 1145.315,A -85,B 0,C 180,E1 11012.158,E2 11012.158} C_VEL
LIN {X 0,Y 282.799,Z 1127.117,A -85,B 0,C 180,E1 11010.215,E2 11010.215} C_VEL
LIN {X 0,Y 291.002,Z 1107.927,A -85,B 0,C 180,E1 11008.616,E2 11008.616} C_VEL
LIN {X 0,Y 298.668,Z 1087.582,A -85,B 0,C 180,E1 11007.299,E2 11007.299} C_VEL
LIN {X 0,Y 305.46,Z 1066.373,A -85,B 0,C 180,E1 11006.253,E2 11006.253} C_VEL
LIN {X 0,Y 310.973,Z 1044.027,A -85,B 0,C 180,E1 11005.399,E2 11005.399} C_VEL
LIN {X 0,Y 314.955,Z 1021.529,A -85,B 0,C 180,E1 11004.728,E2 11004.728} C_VEL
LIN {X 0,Y 317.671,Z 996.585,A -85,B 0,C 180,E1 11004.157,E2 11004.157} C_VEL
LIN {X 0,Y 329.725,Z 852.466,A -85,B 0,C 180,E1 11001.246,E2 11001.246} C_VEL
LIN {X 0,Y 324.929,Z 841.036,A -85,B 0,C 180,E1 10998.385,E2 10998.385} C_VEL
LIN {X 0,Y 320.474,Z 830.743,A -85,B 0,C 180,E1 10995.239,E2 10995.239} C_VEL
LIN {X 0,Y 316.41,Z 821.68,A -85,B 0,C 180,E1 10991.668,E2 10991.668} C_VEL
LIN {X 0,Y 313.622,Z 815.525,A -85,B 0,C 180,E1 10988.433,E2 10988.433} C_VEL
LIN {X 0,Y 311.922,Z 811.628,A -85,B 0,C 180,E1 10985.703,E2 10985.703} C_VEL
LIN {X 0,Y 309.895,Z 809.428,A -85,B 0,C 180,E1 10979.075,E2 10979.075} C_VEL
LIN {X 0,Y 310.491,Z 810.419,A -85,B 0,C 180,E1 10974.826,E2 10974.826} C_VEL
LIN {X 0,Y 312.048,Z 811.961,A -85,B 0,C 180,E1 10971.524,E2 10971.524} C_VEL
LIN {X 0,Y 314.663,Z 816.307,A -85,B 0,C 180,E1 10967.894,E2 10967.894} C_VEL
LIN {X 0,Y 318.326,Z 822.271,A -85,B 0,C 180,E1 10964.328,E2 10964.328} C_VEL
LIN {X 0,Y 321.549,Z 827.57,A -85,B 0,C 180,E1 10961.836,E2 10961.836} C_VEL
LIN {X 0,Y 325.687,Z 834.449,A -85,B 0,C 180,E1 10959.138,E2 10959.138} C_VEL
LIN {X 0,Y 329.745,Z 841.817,A -85,B 0,C 180,E1 10956.82,E2 10956.82} C_VEL
LIN {X 0,Y 320.219,Z 954.883,A -85,B 0,C 180,E1 10954.514,E2 10954.514} C_VEL
LIN {X 0,Y 317.87,Z 976.915,A -85,B 0,C 180,E1 10953.846,E2 10953.846} C_VEL
LIN {X 0,Y 314.24,Z 998.564,A -85,B 0,C 180,E1 10952.947,E2 10952.947} C_VEL
LIN {X 0,Y 309.588,Z 1019.085,A -85,B 0,C 180,E1 10951.844,E2 10951.844} C_VEL
LIN {X 0,Y 303.835,Z 1038.911,A -85,B 0,C 180,E1 10950.504,E2 10950.504} C_VEL
LIN {X 0,Y 297.145,Z 1057.853,A -85,B 0,C 180,E1 10948.908,E2 10948.908} C_VEL
LIN {X 0,Y 289.62,Z 1076.112,A -85,B 0,C 180,E1 10947.023,E2 10947.023} C_VEL
LIN {X 0,Y 281.37,Z 1093.484,A -85,B 0,C 180,E1 10944.814,E2 10944.814} C_VEL
LIN {X 0,Y 272.828,Z 1109.322,A -85,B 0,C 180,E1 10942.333,E2 10942.333} C_VEL
LIN {X 0,Y 263.601,Z 1124.827,A -85,B 0,C 180,E1 10939.34,E2 10939.34} C_VEL
LIN {X 0,Y 254.467,Z 1138.865,A -85,B 0,C 180,E1 10935.974,E2 10935.974} C_VEL
LIN {X 0,Y 245.607,Z 1151.349,A -85,B 0,C 180,E1 10932.19,E2 10932.19} C_VEL
LIN {X 0,Y 237.317,Z 1162.446,A -85,B 0,C 180,E1 10927.96,E2 10927.96} C_VEL
LIN {X 0,Y 229.806,Z 1172.185,A -85,B 0,C 180,E1 10923.243,E2 10923.243} C_VEL
LIN {X 0,Y 223.347,Z 1180.398,A -85,B 0,C 180,E1 10918.037,E2 10918.037} C_VEL
LIN {X 0,Y 218.365,Z 1186.81,A -85,B 0,C 180,E1 10912.62,E2 10912.62} C_VEL
LIN {X 0,Y 214.704,Z 1191.84,A -85,B 0,C 180,E1 10906.781,E2 10906.781} C_VEL
LIN {X 0,Y 212.595,Z 1195.111,A -85,B 0,C 180,E1 10901.118,E2 10901.118} C_VEL
LIN {X 0,Y 211.493,Z 1196.959,A -85,B 0,C 180,E1 10895.425,E2 10895.425} C_VEL
LIN {X 0,Y 211.221,Z 1197.611,A -85,B 0,C 180,E1 10890,E2 10890} C_VEL
LIN {X 0,Y 211.488,Z 1196.989,A -85,B 0,C 180,E1 10884.574,E2 10884.574} C_VEL
LIN {X 0,Y 212.582,Z 1195.18,A -85,B 0,C 180,E1 10878.882,E2 10878.882} C_VEL
LIN {X 0,Y 214.671,Z 1191.927,A -85,B 0,C 180,E1 10873.216,E2 10873.216} C_VEL
LIN {X 0,Y 218.313,Z 1186.935,A -85,B 0,C 180,E1 10867.375,E2 10867.375} C_VEL
LIN {X 0,Y 223.368,Z 1180.441,A -85,B 0,C 180,E1 10861.864,E2 10861.864} C_VEL
LIN {X 0,Y 229.884,Z 1172.176,A -85,B 0,C 180,E1 10856.625,E2 10856.625} C_VEL
LIN {X 0,Y 237.213,Z 1162.68,A -85,B 0,C 180,E1 10852.019,E2 10852.019} C_VEL
LIN {X 0,Y 245.968,Z 1150.969,A -85,B 0,C 180,E1 10847.564,E2 10847.564} C_VEL
LIN {X 0,Y 254.86,Z 1138.418,A -85,B 0,C 180,E1 10843.793,E2 10843.793} C_VEL
LIN {X 0,Y 264.036,Z 1124.327,A -85,B 0,C 180,E1 10840.436,E2 10840.436} C_VEL
LIN {X 0,Y 272.995,Z 1109.239,A -85,B 0,C 180,E1 10837.541,E2 10837.541} C_VEL
LIN {X 0,Y 281.419,Z 1093.649,A -85,B 0,C 180,E1 10835.099,E2 10835.099} C_VEL
LIN {X 0,Y 289.487,Z 1076.685,A -85,B 0,C 180,E1 10832.937,E2 10832.937} C_VEL
LIN {X 0,Y 297.015,Z 1058.547,A -85,B 0,C 180,E1 10831.051,E2 10831.051} C_VEL
LIN {X 0,Y 303.714,Z 1039.78,A -85,B 0,C 180,E1 10829.456,E2 10829.456} C_VEL
LIN {X 0,Y 309.46,Z 1020.063,A -85,B 0,C 180,E1 10828.112,E2 10828.112} C_VEL
LIN {X 0,Y 314.314,Z 998.912,A -85,B 0,C 180,E1 10826.966,E2 10826.966} C_VEL
LIN {X 0,Y 317.936,Z 977.568,A -85,B 0,C 180,E1 10826.075,E2 10826.075} C_VEL
LIN {X 0,Y 320.277,Z 955.866,A -85,B 0,C 180,E1 10825.41,E2 10825.41} C_VEL
LIN {X 0,Y 326.746,Z 878.314,A -85,B 0,C 180,E1 10823.799,E2 10823.799} C_VEL
LIN {X 0,Y 329.895,Z 841.826,A -85,B 0,C 180,E1 10823.077,E2 10823.077} C_VEL
LIN {X 0,Y 324.937,Z 832.976,A -85,B 0,C 180,E1 10820.202,E2 10820.202} C_VEL
LIN {X 0,Y 320.138,Z 825.002,A -85,B 0,C 180,E1 10816.886,E2 10816.886} C_VEL
LIN {X 0,Y 319.114,Z 823.478,A -85,B 0,C 180,E1 10816.086,E2 10816.086} C_VEL
LIN {X 0,Y 317.541,Z 822.063,A -85,B 0,C 180,E1 10814.844,E2 10814.844} C_VEL
LIN {X 0,Y 314.939,Z 822.337,A -85,B 0,C 180,E1 10812.761,E2 10812.761} C_VEL
LIN {X 0,Y 312.641,Z 822.718,A -85,B 0,C 180,E1 10810.527,E2 10810.527} C_VEL
LIN {X 0,Y 312.025,Z 822.099,A -85,B 0,C 180,E1 10809.716,E2 10809.716} C_VEL
LIN {X 0,Y 310.831,Z 819.509,A -85,B 0,C 180,E1 10807.579,E2 10807.579} C_VEL
LIN {X 0,Y 309.146,Z 817.652,A -85,B 0,C 180,E1 10801.298,E2 10801.298} C_VEL
LIN {X 0,Y 310.203,Z 819.049,A -85,B 0,C 180,E1 10796.119,E2 10796.119} C_VEL
LIN {X 0,Y 311.082,Z 819.94,A -85,B 0,C 180,E1 10794.375,E2 10794.375} C_VEL
LIN {X 0,Y 312.556,Z 823.414,A -85,B 0,C 180,E1 10791.909,E2 10791.909} C_VEL
LIN {X 0,Y 315.143,Z 829.365,A -85,B 0,C 180,E1 10788.749,E2 10788.749} C_VEL
LIN {X 0,Y 319.31,Z 839.191,A -85,B 0,C 180,E1 10784.936,E2 10784.936} C_VEL
LIN {X 0,Y 323.547,Z 849.364,A -85,B 0,C 180,E1 10781.86,E2 10781.86} C_VEL
LIN {X 0,Y 326.526,Z 857.053,A -85,B 0,C 180,E1 10779.962,E2 10779.962} C_VEL
LIN {X 0,Y 312.894,Z 1012.242,A -85,B 0,C 180,E1 10776.838,E2 10776.838} C_VEL
LIN {X 0,Y 309.34,Z 1034.602,A -85,B 0,C 180,E1 10776.231,E2 10776.231} C_VEL
LIN {X 0,Y 303.994,Z 1057.896,A -85,B 0,C 180,E1 10775.422,E2 10775.422} C_VEL
LIN {X 0,Y 297.896,Z 1078.328,A -85,B 0,C 180,E1 10774.534,E2 10774.534} C_VEL
LIN {X 0,Y 290.299,Z 1099.064,A -85,B 0,C 180,E1 10773.349,E2 10773.349} C_VEL
LIN {X 0,Y 281.833,Z 1119.05,A -85,B 0,C 180,E1 10771.846,E2 10771.846} C_VEL
LIN {X 0,Y 272.881,Z 1137.89,A -85,B 0,C 180,E1 10770.032,E2 10770.032} C_VEL
LIN {X 0,Y 263.4,Z 1155.78,A -85,B 0,C 180,E1 10767.83,E2 10767.83} C_VEL
LIN {X 0,Y 253.193,Z 1173.482,A -85,B 0,C 180,E1 10765.068,E2 10765.068} C_VEL
LIN {X 0,Y 243.617,Z 1189.149,A -85,B 0,C 180,E1 10761.998,E2 10761.998} C_VEL
LIN {X 0,Y 234.156,Z 1203.905,A -85,B 0,C 180,E1 10758.351,E2 10758.351} C_VEL
LIN {X 0,Y 225.005,Z 1217.996,A -85,B 0,C 180,E1 10753.956,E2 10753.956} C_VEL
LIN {X 0,Y 217.156,Z 1230.371,A -85,B 0,C 180,E1 10749.107,E2 10749.107} C_VEL
LIN {X 0,Y 210.453,Z 1241.793,A -85,B 0,C 180,E1 10743.442,E2 10743.442} C_VEL
LIN {X 0,Y 205.763,Z 1251.12,A -85,B 0,C 180,E1 10737.491,E2 10737.491} C_VEL
LIN {X 0,Y 202.935,Z 1258.948,A -85,B 0,C 180,E1 10731.079,E2 10731.079} C_VEL
LIN {X 0,Y 202.011,Z 1264.457,A -85,B 0,C 180,E1 10725.172,E2 10725.172} C_VEL
LIN {X 0,Y 202.25,Z 1268.016,A -85,B 0,C 180,E1 10719.676,E2 10719.676} C_VEL
LIN {X 0,Y 202.863,Z 1269.927,A -85,B 0,C 180,E1 10715.09,E2 10715.09} C_VEL
LIN {X 0,Y 203.255,Z 1270.69,A -85,B 0,C 180,E1 10710.846,E2 10710.846} C_VEL
LIN {X 0,Y 203.066,Z 1270.391,A -85,B 0,C 180,E1 10706.613,E2 10706.613} C_VEL
LIN {X 0,Y 202.417,Z 1268.74,A -85,B 0,C 180,E1 10701.764,E2 10701.764} C_VEL
LIN {X 0,Y 202.006,Z 1265.861,A -85,B 0,C 180,E1 10696.84,E2 10696.84} C_VEL
LIN {X 0,Y 202.449,Z 1261.061,A -85,B 0,C 180,E1 10690.977,E2 10690.977} C_VEL
